LIN {X 0,Y 310.097,Z 794.889,A -85,B 0,C 180,E1 -20725.805,E2 -20725.805} C_VEL
LIN {X 0,Y 313.218,Z 774.353,A -85,B 0,C 180,E1 -20728.091,E2 -20728.091} C_VEL
LIN {X 0,Y 316.543,Z 751.825,A -85,B 0,C 180,E1 -20730.149,E2 -20730.149} C_VEL
LIN {X 0,Y 319.689,Z 728.685,A -85,B 0,C 180,E1 -20731.857,E2 -20731.857} C_VEL
LIN {X 0,Y 322.597,Z 704.405,A -85,B 0,C 180,E1 -20733.252,E2 -20733.252} C_VEL
LIN {X 0,Y 324.402,Z 688.186,A -85,B 0,C 180,E1 -20734.016,E2 -20734.016} C_VEL
LIN {X 0,Y 325.636,Z 688.059,A -85,B 0,C 180,E1 -20734.348,E2 -20734.348} C_VEL
LIN {X 0,Y 327.891,Z 685.502,A -85,B 0,C 180,E1 -20734.741,E2 -20734.741} C_VEL
LIN {X 0,Y 331.75,Z 678.48,A -85,B 0,C 180,E1 -20735.173,E2 -20735.173} C_VEL
LIN {X 0,Y 336.333,Z 667.667,A -85,B 0,C 180,E1 -20735.483,E2 -20735.483} C_VEL
LIN {X 0,Y 339.475,Z 663.92,A -85,B 0,C 180,E1 -20735.988,E2 -20735.988} C_VEL
LIN {X 0,Y 343.394,Z 656.895,A -85,B 0,C 180,E1 -20736.429,E2 -20736.429} C_VEL
LIN {X 0,Y 348.297,Z 645.248,A -85,B 0,C 180,E1 -20736.772,E2 -20736.772} C_VEL
LIN {X 0,Y 349.24,Z 643.212,A -85,B 0,C 180,E1 -20736.856,E2 -20736.856} C_VEL
LIN {X 0,Y 353.089,Z 637.648,A -85,B 0,C 180,E1 -20737.379,E2 -20737.379} C_VEL
LIN {X 0,Y 357.645,Z 628.586,A -85,B 0,C 180,E1 -20737.818,E2 -20737.818} C_VEL
LIN {X 0,Y 363.002,Z 615.103,A -85,B 0,C 180,E1 -20738.174,E2 -20738.174} C_VEL
LIN {X 0,Y 367.492,Z 607.691,A -85,B 0,C 180,E1 -20738.703,E2 -20738.703} C_VEL
LIN {X 0,Y 372.393,Z 596.823,A -85,B 0,C 180,E1 -20739.123,E2 -20739.123} C_VEL
LIN {X 0,Y 375.613,Z 588.328,A -85,B 0,C 180,E1 -20739.332,E2 -20739.332} C_VEL
LIN {X 0,Y 368.648,Z 640.972,A -85,B 0,C 180,E1 -20740.837,E2 -20740.837} C_VEL
LIN {X 0,Y 363.114,Z 683.795,A -85,B 0,C 180,E1 -20742.409,E2 -20742.409} C_VEL
LIN {X 0,Y 360.052,Z 705.878,A -85,B 0,C 180,E1 -20743.431,E2 -20743.431} C_VEL
LIN {X 0,Y 356.301,Z 726.402,A -85,B 0,C 180,E1 -20744.651,E2 -20744.651} C_VEL
LIN {X 0,Y 351.864,Z 746.01,A -85,B 0,C 180,E1 -20746.102,E2 -20746.102} C_VEL
LIN {X 0,Y 346.634,Z 765.549,A -85,B 0,C 180,E1 -20747.881,E2 -20747.881} C_VEL
LIN {X 0,Y 340.825,Z 784.337,A -85,B 0,C 180,E1 -20749.97,E2 -20749.97} C_VEL
LIN {X 0,Y 334.834,Z 801.656,A -85,B 0,C 180,E1 -20752.312,E2 -20752.312} C_VEL
LIN {X 0,Y 328.814,Z 817.581,A -85,B 0,C 180,E1 -20754.919,E2 -20754.919} C_VEL
LIN {X 0,Y 322.895,Z 832.224,A -85,B 0,C 180,E1 -20757.817,E2 -20757.817} C_VEL
LIN {X 0,Y 317.342,Z 845.359,A -85,B 0,C 180,E1 -20760.972,E2 -20760.972} C_VEL
LIN {X 0,Y 312.298,Z 857,A -85,B 0,C 180,E1 -20764.391,E2 -20764.391} C_VEL
LIN {X 0,Y 307.902,Z 867.134,A -85,B 0,C 180,E1 -20768.071,E2 -20768.071} C_VEL
LIN {X 0,Y 304.295,Z 875.703,A -85,B 0,C 180,E1 -20772.008,E2 -20772.008} C_VEL
LIN {X 0,Y 301.659,Z 882.344,A -85,B 0,C 180,E1 -20775.997,E2 -20775.997} C_VEL
LIN {X 0,Y 299.834,Z 887.403,A -85,B 0,C 180,E1 -20780.208,E2 -20780.208} C_VEL
LIN {X 0,Y 298.86,Z 890.521,A -85,B 0,C 180,E1 -20784.239,E2 -20784.239} C_VEL
LIN {X 0,Y 298.446,Z 892.023,A -85,B 0,C 180,E1 -20788.08,E2 -20788.08} C_VEL
LIN {X 0,Y 298.441,Z 892.036,A -85,B 0,C 180,E1 -20791.92,E2 -20791.92} C_VEL
LIN {X 0,Y 298.847,Z 890.585,A -85,B 0,C 180,E1 -20795.761,E2 -20795.761} C_VEL
LIN {X 0,Y 299.808,Z 887.52,A -85,B 0,C 180,E1 -20799.793,E2 -20799.793} C_VEL
LIN {X 0,Y 301.515,Z 882.791,A -85,B 0,C 180,E1 -20803.814,E2 -20803.814} C_VEL
LIN {X 0,Y 303.952,Z 876.657,A -85,B 0,C 180,E1 -20807.616,E2 -20807.616} C_VEL
LIN {X 0,Y 307.265,Z 868.804,A -85,B 0,C 180,E1 -20811.375,E2 -20811.375} C_VEL
LIN {X 0,Y 311.499,Z 859.044,A -85,B 0,C 180,E1 -20815.069,E2 -20815.069} C_VEL
LIN {X 0,Y 316.674,Z 847.142,A -85,B 0,C 180,E1 -20818.681,E2 -20818.681} C_VEL
LIN {X 0,Y 322.136,Z 834.333,A -85,B 0,C 180,E1 -20821.848,E2 -20821.848} C_VEL
LIN {X 0,Y 327.967,Z 820.047,A -85,B 0,C 180,E1 -20824.758,E2 -20824.758} C_VEL
LIN {X 0,Y 334.223,Z 803.699,A -85,B 0,C 180,E1 -20827.503,E2 -20827.503} C_VEL
LIN {X 0,Y 339.242,Z 789.378,A -85,B 0,C 180,E1 -20829.505,E2 -20829.505} C_VEL
LIN {X 0,Y 340.475,Z 783.625,A -85,B 0,C 180,E1 -20830.359,E2 -20830.359} C_VEL
LIN {X 0,Y 340.769,Z 769.373,A -85,B 0,C 180,E1 -20832.726,E2 -20832.726} C_VEL
LIN {X 0,Y 341.959,Z 763.048,A -85,B 0,C 180,E1 -20833.483,E2 -20833.483} C_VEL
LIN {X 0,Y 346.995,Z 744.339,A -85,B 0,C 180,E1 -20835.143,E2 -20835.143} C_VEL
LIN {X 0,Y 351.352,Z 725.232,A -85,B 0,C 180,E1 -20836.526,E2 -20836.526} C_VEL
LIN {X 0,Y 355.11,Z 704.688,A -85,B 0,C 180,E1 -20837.724,E2 -20837.724} C_VEL
LIN {X 0,Y 358.615,Z 679.329,A -85,B 0,C 180,E1 -20838.859,E2 -20838.859} C_VEL
LIN {X 0,Y 364.283,Z 637.626,A -85,B 0,C 180,E1 -20840.362,E2 -20840.362} C_VEL
LIN {X 0,Y 371.135,Z 586.782,A -85,B 0,C 180,E1 -20841.799,E2 -20841.799} C_VEL
LIN {X 0,Y 377.109,Z 533.395,A -85,B 0,C 180,E1 -20843.058,E2 -20843.058} C_VEL
LIN {X 0,Y 381.368,Z 483.071,A -85,B 0,C 180,E1 -20844.053,E2 -20844.053} C_VEL
LIN {X 0,Y 384.825,Z 436.662,A -85,B 0,C 180,E1 -20844.887,E2 -20844.887} C_VEL
LIN {X 0,Y 391.487,Z 407.522,A -85,B 0,C 180,E1 -20845.872,E2 -20845.872} C_VEL
LIN {X 0,Y 386.519,Z 392.199,A -85,B 0,C 180,E1 -20848.67,E2 -20848.67} C_VEL
LIN {X 0,Y 381.381,Z 378.048,A -85,B 0,C 180,E1 -20851.67,E2 -20851.67} C_VEL
LIN {X 0,Y 376.23,Z 365.361,A -85,B 0,C 180,E1 -20854.835,E2 -20854.835} C_VEL
LIN {X 0,Y 371.348,Z 354.346,A -85,B 0,C 180,E1 -20858.104,E2 -20858.104} C_VEL
LIN {X 0,Y 367.077,Z 345.55,A -85,B 0,C 180,E1 -20861.251,E2 -20861.251} C_VEL
LIN {X 0,Y 364.606,Z 340.77,A -85,B 0,C 180,E1 -20863.265,E2 -20863.265} C_VEL
LIN {X 0,Y 362.517,Z 336.712,A -85,B 0,C 180,E1 -20865.137,E2 -20865.137} C_VEL
LIN {X 0,Y 360.35,Z 332.462,A -85,B 0,C 180,E1 -20867.419,E2 -20867.419} C_VEL
LIN {X 0,Y 357.865,Z 327.689,A -85,B 0,C 180,E1 -20870.511,E2 -20870.511} C_VEL
LIN {X 0,Y 355.935,Z 324.353,A -85,B 0,C 180,E1 -20873.71,E2 -20873.71} C_VEL
LIN {X 0,Y 355.5,Z 322.634,A -85,B 0,C 180,E1 -20874.998,E2 -20874.998} C_VEL
LIN {X 0,Y 354.47,Z 320.986,A -85,B 0,C 180,E1 -20881.455,E2 -20881.455} C_VEL
LIN {X 0,Y 355.671,Z 321.876,A -85,B 0,C 180,E1 -20885.971,E2 -20885.971} C_VEL
LIN {X 0,Y 357.257,Z 323.157,A -85,B 0,C 180,E1 -20888.449,E2 -20888.449} C_VEL
LIN {X 0,Y 359.098,Z 335.798,A -85,B 0,C 180,E1 -20892.871,E2 -20892.871} C_VEL
LIN {X 0,Y 362.564,Z 349.288,A -85,B 0,C 180,E1 -20896.87,E2 -20896.87} C_VEL
LIN {X 0,Y 369.014,Z 369.011,A -85,B 0,C 180,E1 -20901.791,E2 -20901.791} C_VEL
LIN {X 0,Y 372.901,Z 379.636,A -85,B 0,C 180,E1 -20904.052,E2 -20904.052} C_VEL
LIN {X 0,Y 380.695,Z 402.746,A -85,B 0,C 180,E1 -20908.065,E2 -20908.065} C_VEL
LIN {X 0,Y 381.092,Z 404.189,A -85,B 0,C 180,E1 -20908.265,E2 -20908.265} C_VEL
LIN {X 0,Y 363.956,Z 554.058,A -85,B 0,C 180,E1 -20912.157,E2 -20912.157} C_VEL
LIN {X 0,Y 358.565,Z 611.238,A -85,B 0,C 180,E1 -20913.592,E2 -20913.592} C_VEL
LIN {X 0,Y 355.678,Z 653.164,A -85,B 0,C 180,E1 -20914.491,E2 -20914.491} C_VEL
LIN {X 0,Y 352.117,Z 687.641,A -85,B 0,C 180,E1 -20915.473,E2 -20915.473} C_VEL
LIN {X 0,Y 347.408,Z 721.446,A -85,B 0,C 180,E1 -20916.703,E2 -20916.703} C_VEL
LIN {X 0,Y 342.681,Z 750.705,A -85,B 0,C 180,E1 -20918.083,E2 -20918.083} C_VEL
LIN {X 0,Y 337.211,Z 780.861,A -85,B 0,C 180,E1 -20919.828,E2 -20919.828} C_VEL
LIN {X 0,Y 331.507,Z 809.252,A -85,B 0,C 180,E1 -20921.841,E2 -20921.841} C_VEL
LIN {X 0,Y 327.245,Z 827.893,A -85,B 0,C 180,E1 -20923.475,E2 -20923.475} C_VEL
LIN {X 0,Y 322.518,Z 845.852,A -85,B 0,C 180,E1 -20925.396,E2 -20925.396} C_VEL
LIN {X 0,Y 317.602,Z 862.404,A -85,B 0,C 180,E1 -20927.523,E2 -20927.523} C_VEL
LIN {X 0,Y 312.385,Z 878.87,A -85,B 0,C 180,E1 -20930.076,E2 -20930.076} C_VEL
LIN {X 0,Y 307.204,Z 894.344,A -85,B 0,C 180,E1 -20932.977,E2 -20932.977} C_VEL
LIN {X 0,Y 302.284,Z 908.668,A -85,B 0,C 180,E1 -20936.241,E2 -20936.241} C_VEL
LIN {X 0,Y 297.991,Z 921.531,A -85,B 0,C 180,E1 -20939.781,E2 -20939.781} C_VEL
LIN {X 0,Y 294.466,Z 932.94,A -85,B 0,C 180,E1 -20943.588,E2 -20943.588} C_VEL
LIN {X 0,Y 291.816,Z 942.875,A -85,B 0,C 180,E1 -20947.69,E2 -20947.69} C_VEL
LIN {X 0,Y 290.161,Z 951.193,A -85,B 0,C 180,E1 -20952.007,E2 -20952.007} C_VEL
LIN {X 0,Y 289.494,Z 957.489,A -85,B 0,C 180,E1 -20956.213,E2 -20956.213} C_VEL
LIN {X 0,Y 289.553,Z 962.147,A -85,B 0,C 180,E1 -20960.459,E2 -20960.459} C_VEL
LIN {X 0,Y 289.9,Z 965.745,A -85,B 0,C 180,E1 -20964.657,E2 -20964.657} C_VEL
LIN {X 0,Y 290.044,Z 968.016,A -85,B 0,C 180,E1 -20968.222,E2 -20968.222} C_VEL
LIN {X 0,Y 289.94,Z 968.994,A -85,B 0,C 180,E1 -20971.383,E2 -20971.383} C_VEL
LIN {X 0,Y 289.558,Z 968.983,A -85,B 0,C 180,E1 -20974.754,E2 -20974.754} C_VEL
LIN {X 0,Y 289.099,Z 967.8,A -85,B 0,C 180,E1 -20978.553,E2 -20978.553} C_VEL
LIN {X 0,Y 288.987,Z 964.607,A -85,B 0,C 180,E1 -20983.404,E2 -20983.404} C_VEL
LIN {X 0,Y 289.757,Z 960.148,A -85,B 0,C 180,E1 -20987.886,E2 -20987.886} C_VEL
LIN {X 0,Y 292.21,Z 953.138,A -85,B 0,C 180,E1 -20993.173,E2 -20993.173} C_VEL
LIN {X 0,Y 296.428,Z 944.613,A -85,B 0,C 180,E1 -20998.18,E2 -20998.18} C_VEL
LIN {X 0,Y 303.398,Z 933.28,A -85,B 0,C 180,E1 -21003.509,E2 -21003.509} C_VEL
LIN {X 0,Y 312.593,Z 920.465,A -85,B 0,C 180,E1 -21008.401,E2 -21008.401} C_VEL
LIN {X 0,Y 324.233,Z 905.701,A -85,B 0,C 180,E1 -21012.964,E2 -21012.964} C_VEL
LIN {X 0,Y 338.331,Z 889.038,A -85,B 0,C 180,E1 -21017.133,E2 -21017.133} C_VEL
LIN {X 0,Y 354.739,Z 870.663,A -85,B 0,C 180,E1 -21020.817,E2 -21020.817} C_VEL
LIN {X 0,Y 365.018,Z 859.44,A -85,B 0,C 180,E1 -21022.699,E2 -21022.699} C_VEL
LIN {X 0,Y 349.209,Z 872.446,A -85,B 0,C 180,E1 -21025.662,E2 -21025.662} C_VEL
LIN {X 0,Y 335.594,Z 883.653,A -85,B 0,C 180,E1 -21028.972,E2 -21028.972} C_VEL
LIN {X 0,Y 324.384,Z 892.704,A -85,B 0,C 180,E1 -21032.46,E2 -21032.46} C_VEL
LIN {X 0,Y 315.292,Z 899.629,A -85,B 0,C 180,E1 -21036.051,E2 -21036.051} C_VEL
LIN {X 0,Y 308.049,Z 904.537,A -85,B 0,C 180,E1 -21039.677,E2 -21039.677} C_VEL
LIN {X 0,Y 302.172,Z 907.645,A -85,B 0,C 180,E1 -21043.467,E2 -21043.467} C_VEL
LIN {X 0,Y 297.811,Z 908.844,A -85,B 0,C 180,E1 -21047.197,E2 -21047.197} C_VEL
LIN {X 0,Y 294.664,Z 908.287,A -85,B 0,C 180,E1 -21050.917,E2 -21050.917} C_VEL
LIN {X 0,Y 292.468,Z 905.923,A -85,B 0,C 180,E1 -21054.704,E2 -21054.704} C_VEL
LIN {X 0,Y 291.159,Z 901.801,A -85,B 0,C 180,E1 -21058.426,E2 -21058.426} C_VEL
LIN {X 0,Y 290.513,Z 895.812,A -85,B 0,C 180,E1 -21062.17,E2 -21062.17} C_VEL
LIN {X 0,Y 290.44,Z 888.231,A -85,B 0,C 180,E1 -21065.769,E2 -21065.769} C_VEL
LIN {X 0,Y 290.873,Z 878.851,A -85,B 0,C 180,E1 -21069.298,E2 -21069.298} C_VEL
LIN {X 0,Y 291.811,Z 867.931,A -85,B 0,C 180,E1 -21072.668,E2 -21072.668} C_VEL
LIN {X 0,Y 293.234,Z 855.611,A -85,B 0,C 180,E1 -21075.83,E2 -21075.83} C_VEL
LIN {X 0,Y 295.081,Z 841.982,A -85,B 0,C 180,E1 -21078.779,E2 -21078.779} C_VEL
LIN {X 0,Y 297.464,Z 826.09,A -85,B 0,C 180,E1 -21081.7,E2 -21081.7} C_VEL
LIN {X 0,Y 300.213,Z 808.748,A -85,B 0,C 180,E1 -21084.393,E2 -21084.393} C_VEL
LIN {X 0,Y 303.242,Z 789.904,A -85,B 0,C 180,E1 -21086.855,E2 -21086.855} C_VEL
LIN {X 0,Y 306.442,Z 769.276,A -85,B 0,C 180,E1 -21089.09,E2 -21089.09} C_VEL
LIN {X 0,Y 309.807,Z 746.584,A -85,B 0,C 180,E1 -21091.091,E2 -21091.091} C_VEL
LIN {X 0,Y 313.021,Z 722.706,A -85,B 0,C 180,E1 -21092.782,E2 -21092.782} C_VEL
LIN {X 0,Y 314.397,Z 711.79,A -85,B 0,C 180,E1 -21093.435,E2 -21093.435} C_VEL
LIN {X 0,Y 315.558,Z 711.842,A -85,B 0,C 180,E1 -21093.787,E2 -21093.787} C_VEL
LIN {X 0,Y 317.977,Z 709.611,A -85,B 0,C 180,E1 -21094.255,E2 -21094.255} C_VEL
LIN {X 0,Y 321.775,Z 703.882,A -85,B 0,C 180,E1 -21094.738,E2 -21094.738} C_VEL
LIN {X 0,Y 326.016,Z 695.125,A -85,B 0,C 180,E1 -21095.091,E2 -21095.091} C_VEL
LIN {X 0,Y 329.867,Z 690.849,A -85,B 0,C 180,E1 -21095.724,E2 -21095.724} C_VEL
LIN {X 0,Y 333.975,Z 683.923,A -85,B 0,C 180,E1 -21096.196,E2 -21096.196} C_VEL
LIN {X 0,Y 338.441,Z 674.02,A -85,B 0,C 180,E1 -21096.514,E2 -21096.514} C_VEL
LIN {X 0,Y 339.39,Z 672.118,A -85,B 0,C 180,E1 -21096.6,E2 -21096.6} C_VEL
LIN {X 0,Y 343.392,Z 666.592,A -85,B 0,C 180,E1 -21097.145,E2 -21097.145} C_VEL
LIN {X 0,Y 348.05,Z 657.692,A -85,B 0,C 180,E1 -21097.589,E2 -21097.589} C_VEL
LIN {X 0,Y 352.501,Z 647.411,A -85,B 0,C 180,E1 -21097.888,E2 -21097.888} C_VEL
LIN {X 0,Y 357.058,Z 640.454,A -85,B 0,C 180,E1 -21098.439,E2 -21098.439} C_VEL
LIN {X 0,Y 362.014,Z 630.337,A -85,B 0,C 180,E1 -21098.87,E2 -21098.87} C_VEL
LIN {X 0,Y 366.643,Z 618.897,A -85,B 0,C 180,E1 -21099.159,E2 -21099.159} C_VEL
LIN {X 0,Y 360.03,Z 667.651,A -85,B 0,C 180,E1 -21100.794,E2 -21100.794} C_VEL
LIN {X 0,Y 355.595,Z 700.826,A -85,B 0,C 180,E1 -21102.189,E2 -21102.189} C_VEL
LIN {X 0,Y 351.844,Z 722.205,A -85,B 0,C 180,E1 -21103.388,E2 -21103.388} C_VEL
LIN {X 0,Y 347.315,Z 742.561,A -85,B 0,C 180,E1 -21104.826,E2 -21104.826} C_VEL
LIN {X 0,Y 342.182,Z 761.879,A -85,B 0,C 180,E1 -21106.516,E2 -21106.516} C_VEL
LIN {X 0,Y 336.449,Z 780.451,A -85,B 0,C 180,E1 -21108.497,E2 -21108.497} C_VEL
LIN {X 0,Y 330.364,Z 797.932,A -85,B 0,C 180,E1 -21110.76,E2 -21110.76} C_VEL
LIN {X 0,Y 324.065,Z 814.382,A -85,B 0,C 180,E1 -21113.343,E2 -21113.343} C_VEL
LIN {X 0,Y 317.926,Z 829.258,A -85,B 0,C 180,E1 -21116.174,E2 -21116.174} C_VEL
LIN {X 0,Y 311.925,Z 843.014,A -85,B 0,C 180,E1 -21119.357,E2 -21119.357} C_VEL
LIN {X 0,Y 306.423,Z 855.219,A -85,B 0,C 180,E1 -21122.817,E2 -21122.817} C_VEL
LIN {X 0,Y 301.577,Z 865.858,A -85,B 0,C 180,E1 -21126.555,E2 -21126.555} C_VEL
LIN {X 0,Y 297.526,Z 874.902,A -85,B 0,C 180,E1 -21130.567,E2 -21130.567} C_VEL
LIN {X 0,Y 294.517,Z 881.994,A -85,B 0,C 180,E1 -21134.644,E2 -21134.644} C_VEL
LIN {X 0,Y 292.358,Z 887.482,A -85,B 0,C 180,E1 -21138.958,E2 -21138.958} C_VEL
LIN {X 0,Y 291.105,Z 891.11,A -85,B 0,C 180,E1 -21143.293,E2 -21143.293} C_VEL
LIN {X 0,Y 290.551,Z 892.885,A -85,B 0,C 180,E1 -21147.436,E2 -21147.436} C_VEL
LIN {X 0,Y 290.477,Z 893.097,A -85,B 0,C 180,E1 -21151.381,E2 -21151.381} C_VEL
LIN {X 0,Y 290.873,Z 891.794,A -85,B 0,C 180,E1 -21155.523,E2 -21155.523} C_VEL
LIN {X 0,Y 291.835,Z 888.902,A -85,B 0,C 180,E1 -21159.665,E2 -21159.665} C_VEL
LIN {X 0,Y 293.569,Z 884.354,A -85,B 0,C 180,E1 -21163.793,E2 -21163.793} C_VEL
LIN {X 0,Y 296.202,Z 878.044,A -85,B 0,C 180,E1 -21167.89,E2 -21167.89} C_VEL
LIN {X 0,Y 299.836,Z 869.83,A -85,B 0,C 180,E1 -21171.931,E2 -21171.931} C_VEL
LIN {X 0,Y 304.281,Z 860.081,A -85,B 0,C 180,E1 -21175.706,E2 -21175.706} C_VEL
LIN {X 0,Y 309.693,Z 848.18,A -85,B 0,C 180,E1 -21179.39,E2 -21179.39} C_VEL
LIN {X 0,Y 315.388,Z 835.383,A -85,B 0,C 180,E1 -21182.613,E2 -21182.613} C_VEL
LIN {X 0,Y 321.456,Z 821.111,A -85,B 0,C 180,E1 -21185.568,E2 -21185.568} C_VEL
LIN {X 0,Y 327.943,Z 804.743,A -85,B 0,C 180,E1 -21188.35,E2 -21188.35} C_VEL
LIN {X 0,Y 334.1,Z 787.79,A -85,B 0,C 180,E1 -21190.725,E2 -21190.725} C_VEL
LIN {X 0,Y 339.952,Z 769.852,A -85,B 0,C 180,E1 -21192.799,E2 -21192.799} C_VEL
LIN {X 0,Y 341.959,Z 763.048,A -85,B 0,C 180,E1 -21193.483,E2 -21193.483} C_VEL
LIN {X 0,Y 343.111,Z 756.729,A -85,B 0,C 180,E1 -21194.213,E2 -21194.213} C_VEL
LIN {X 0,Y 343.287,Z 740.949,A -85,B 0,C 180,E1 -21196.295,E2 -21196.295} C_VEL
LIN {X 0,Y 344.169,Z 734.277,A -85,B 0,C 180,E1 -21196.932,E2 -21196.932} C_VEL
LIN {X 0,Y 348.496,Z 713.392,A -85,B 0,C 180,E1 -21198.268,E2 -21198.268} C_VEL
LIN {X 0,Y 351.931,Z 691.641,A -85,B 0,C 180,E1 -21199.351,E2 -21199.351} C_VEL
LIN {X 0,Y 357.689,Z 649.532,A -85,B 0,C 180,E1 -21200.974,E2 -21200.974} C_VEL
LIN {X 0,Y 364.593,Z 600.878,A -85,B 0,C 180,E1 -21202.435,E2 -21202.435} C_VEL
LIN {X 0,Y 370.767,Z 550.378,A -85,B 0,C 180,E1 -21203.692,E2 -21203.692} C_VEL
LIN {X 0,Y 375.515,Z 499.905,A -85,B 0,C 180,E1 -21204.738,E2 -21204.738} C_VEL
LIN {X 0,Y 380.163,Z 439.411,A -85,B 0,C 180,E1 -21205.836,E2 -21205.836} C_VEL
LIN {X 0,Y 386.666,Z 411.148,A -85,B 0,C 180,E1 -21206.777,E2 -21206.777} C_VEL
LIN {X 0,Y 381.926,Z 396.352,A -85,B 0,C 180,E1 -21209.563,E2 -21209.563} C_VEL
LIN {X 0,Y 376.863,Z 382.161,A -85,B 0,C 180,E1 -21212.677,E2 -21212.677} C_VEL
LIN {X 0,Y 372.149,Z 370.419,A -85,B 0,C 180,E1 -21215.727,E2 -21215.727} C_VEL
LIN {X 0,Y 367.922,Z 360.719,A -85,B 0,C 180,E1 -21218.685,E2 -21218.685} C_VEL
LIN {X 0,Y 364.04,Z 352.331,A -85,B 0,C 180,E1 -21221.753,E2 -21221.753} C_VEL
LIN {X 0,Y 361.674,Z 347.588,A -85,B 0,C 180,E1 -21223.786,E2 -21223.786} C_VEL
LIN {X 0,Y 359.895,Z 343.923,A -85,B 0,C 180,E1 -21225.52,E2 -21225.52} C_VEL
LIN {X 0,Y 357.988,Z 339.875,A -85,B 0,C 180,E1 -21227.744,E2 -21227.744} C_VEL
LIN {X 0,Y 355.585,Z 335.237,A -85,B 0,C 180,E1 -21230.777,E2 -21230.777} C_VEL
LIN {X 0,Y 353.736,Z 331.636,A -85,B 0,C 180,E1 -21234.159,E2 -21234.159} C_VEL
LIN {X 0,Y 353.406,Z 330.304,A -85,B 0,C 180,E1 -21235.294,E2 -21235.294} C_VEL
LIN {X 0,Y 352.685,Z 328.775,A -85,B 0,C 180,E1 -21241.625,E2 -21241.625} C_VEL
LIN {X 0,Y 354.065,Z 329.807,A -85,B 0,C 180,E1 -21246.323,E2 -21246.323} C_VEL
LIN {X 0,Y 355.236,Z 330.811,A -85,B 0,C 180,E1 -21248.172,E2 -21248.172} C_VEL
LIN {X 0,Y 356.963,Z 342.871,A -85,B 0,C 180,E1 -21252.374,E2 -21252.374} C_VEL
LIN {X 0,Y 360.086,Z 356.086,A -85,B 0,C 180,E1 -21256.329,E2 -21256.329} C_VEL
LIN {X 0,Y 366.35,Z 375.856,A -85,B 0,C 180,E1 -21261.285,E2 -21261.285} C_VEL
LIN {X 0,Y 369.886,Z 385.971,A -85,B 0,C 180,E1 -21263.457,E2 -21263.457} C_VEL
LIN {X 0,Y 376.95,Z 407.665,A -85,B 0,C 180,E1 -21267.271,E2 -21267.271} C_VEL
LIN {X 0,Y 356.204,Z 579.083,A -85,B 0,C 180,E1 -21271.835,E2 -21271.835} C_VEL
LIN {X 0,Y 351.392,Z 648.87,A -85,B 0,C 180,E1 -21273.325,E2 -21273.325} C_VEL
LIN {X 0,Y 347.833,Z 683.011,A -85,B 0,C 180,E1 -21274.279,E2 -21274.279} C_VEL
LIN {X 0,Y 343.149,Z 716.179,A -85,B 0,C 180,E1 -21275.459,E2 -21275.459} C_VEL
LIN {X 0,Y 338.014,Z 746.973,A -85,B 0,C 180,E1 -21276.867,E2 -21276.867} C_VEL
LIN {X 0,Y 332.497,Z 776.814,A -85,B 0,C 180,E1 -21278.567,E2 -21278.567} C_VEL
LIN {X 0,Y 326.517,Z 805.796,A -85,B 0,C 180,E1 -21280.585,E2 -21280.585} C_VEL
LIN {X 0,Y 322.047,Z 824.838,A -85,B 0,C 180,E1 -21282.227,E2 -21282.227} C_VEL
LIN {X 0,Y 316.988,Z 843.135,A -85,B 0,C 180,E1 -21284.155,E2 -21284.155} C_VEL
LIN {X 0,Y 311.435,Z 861.14,A -85,B 0,C 180,E1 -21286.475,E2 -21286.475} C_VEL
LIN {X 0,Y 305.778,Z 878.186,A -85,B 0,C 180,E1 -21289.156,E2 -21289.156} C_VEL
LIN {X 0,Y 300.361,Z 893.477,A -85,B 0,C 180,E1 -21292.089,E2 -21292.089} C_VEL
LIN {X 0,Y 295.216,Z 907.713,A -85,B 0,C 180,E1 -21295.39,E2 -21295.39} C_VEL
LIN {X 0,Y 290.74,Z 920.364,A -85,B 0,C 180,E1 -21298.945,E2 -21298.945} C_VEL
LIN {X 0,Y 286.97,Z 931.798,A -85,B 0,C 180,E1 -21302.842,E2 -21302.842} C_VEL
LIN {X 0,Y 284.132,Z 941.659,A -85,B 0,C 180,E1 -21307.007,E2 -21307.007} C_VEL
LIN {X 0,Y 282.324,Z 949.983,A -85,B 0,C 180,E1 -21311.413,E2 -21311.413} C_VEL
LIN {X 0,Y 281.545,Z 956.442,A -85,B 0,C 180,E1 -21315.824,E2 -21315.824} C_VEL
LIN {X 0,Y 281.547,Z 960.921,A -85,B 0,C 180,E1 -21319.979,E2 -21319.979} C_VEL
LIN {X 0,Y 282.01,Z 964.446,A -85,B 0,C 180,E1 -21324.711,E2 -21324.711} C_VEL
LIN {X 0,Y 282.157,Z 966.76,A -85,B 0,C 180,E1 -21328.376,E2 -21328.376} C_VEL
LIN {X 0,Y 281.994,Z 967.796,A -85,B 0,C 180,E1 -21331.829,E2 -21331.829} C_VEL
LIN {X 0,Y 281.58,Z 967.758,A -85,B 0,C 180,E1 -21335.298,E2 -21335.298} C_VEL
LIN {X 0,Y 281.082,Z 966.455,A -85,B 0,C 180,E1 -21339.418,E2 -21339.418} C_VEL
LIN {X 0,Y 281.08,Z 963.184,A -85,B 0,C 180,E1 -21344.419,E2 -21344.419} C_VEL
LIN {X 0,Y 282.123,Z 958.691,A -85,B 0,C 180,E1 -21349.03,E2 -21349.03} C_VEL
LIN {X 0,Y 285.023,Z 951.705,A -85,B 0,C 180,E1 -21354.454,E2 -21354.454} C_VEL
LIN {X 0,Y 290.041,Z 942.875,A -85,B 0,C 180,E1 -21359.764,E2 -21359.764} C_VEL
LIN {X 0,Y 297.987,Z 931.43,A -85,B 0,C 180,E1 -21365.25,E2 -21365.25} C_VEL
LIN {X 0,Y 308.228,Z 918.66,A -85,B 0,C 180,E1 -21370.208,E2 -21370.208} C_VEL
LIN {X 0,Y 320.962,Z 904.077,A -85,B 0,C 180,E1 -21374.754,E2 -21374.754} C_VEL
LIN {X 0,Y 336.752,Z 887.173,A -85,B 0,C 180,E1 -21378.989,E2 -21378.989} C_VEL
LIN {X 0,Y 353.463,Z 870.171,A -85,B 0,C 180,E1 -21382.38,E2 -21382.38} C_VEL
LIN {X 0,Y 355.449,Z 868.133,A -85,B 0,C 180,E1 -21382.756,E2 -21382.756} C_VEL
LIN {X 0,Y 339.797,Z 879.829,A -85,B 0,C 180,E1 -21385.803,E2 -21385.803} C_VEL
LIN {X 0,Y 326.256,Z 889.867,A -85,B 0,C 180,E1 -21389.215,E2 -21389.215} C_VEL
LIN {X 0,Y 315.116,Z 897.821,A -85,B 0,C 180,E1 -21392.811,E2 -21392.811} C_VEL
LIN {X 0,Y 306.095,Z 903.73,A -85,B 0,C 180,E1 -21396.514,E2 -21396.514} C_VEL
LIN {X 0,Y 298.648,Z 907.843,A -85,B 0,C 180,E1 -21400.439,E2 -21400.439} C_VEL
LIN {X 0,Y 292.968,Z 909.937,A -85,B 0,C 180,E1 -21404.358,E2 -21404.358} C_VEL
LIN {X 0,Y 288.828,Z 910.181,A -85,B 0,C 180,E1 -21408.214,E2 -21408.214} C_VEL
LIN {X 0,Y 285.968,Z 908.753,A -85,B 0,C 180,E1 -21411.96,E2 -21411.96} C_VEL
LIN {X 0,Y 283.949,Z 905.358,A -85,B 0,C 180,E1 -21415.961,E2 -21415.961} C_VEL
LIN {X 0,Y 282.868,Z 900.293,A -85,B 0,C 180,E1 -21419.797,E2 -21419.797} C_VEL
LIN {X 0,Y 282.437,Z 893.734,A -85,B 0,C 180,E1 -21423.45,E2 -21423.45} C_VEL
LIN {X 0,Y 282.553,Z 885.362,A -85,B 0,C 180,E1 -21427.115,E2 -21427.115} C_VEL
LIN {X 0,Y 283.163,Z 875.563,A -85,B 0,C 180,E1 -21430.581,E2 -21430.581} C_VEL
LIN {X 0,Y 284.429,Z 862.976,A -85,B 0,C 180,E1 -21434.246,E2 -21434.246} C_VEL
LIN {X 0,Y 286.155,Z 849.601,A -85,B 0,C 180,E1 -21437.488,E2 -21437.488} C_VEL
LIN {X 0,Y 288.324,Z 834.796,A -85,B 0,C 180,E1 -21440.504,E2 -21440.504} C_VEL
LIN {X 0,Y 290.976,Z 818.009,A -85,B 0,C 180,E1 -21443.395,E2 -21443.395} C_VEL
LIN {X 0,Y 293.944,Z 799.899,A -85,B 0,C 180,E1 -21446.028,E2 -21446.028} C_VEL
LIN {X 0,Y 297.289,Z 779.355,A -85,B 0,C 180,E1 -21448.529,E2 -21448.529} C_VEL
LIN {X 0,Y 300.696,Z 757.667,A -85,B 0,C 180,E1 -21450.692,E2 -21450.692} C_VEL
LIN {X 0,Y 304.018,Z 734.908,A -85,B 0,C 180,E1 -21452.53,E2 -21452.53} C_VEL
LIN {X 0,Y 304.579,Z 731.096,A -85,B 0,C 180,E1 -21452.816,E2 -21452.816} C_VEL
LIN {X 0,Y 306.11,Z 730.891,A -85,B 0,C 180,E1 -21453.282,E2 -21453.282} C_VEL
LIN {X 0,Y 308.996,Z 728.323,A -85,B 0,C 180,E1 -21453.82,E2 -21453.82} C_VEL
LIN {X 0,Y 313.01,Z 722.831,A -85,B 0,C 180,E1 -21454.32,E2 -21454.32} C_VEL
LIN {X 0,Y 315.541,Z 718.67,A -85,B 0,C 180,E1 -21454.557,E2 -21454.557} C_VEL
LIN {X 0,Y 319.129,Z 715.537,A -85,B 0,C 180,E1 -21455.205,E2 -21455.205} C_VEL
LIN {X 0,Y 323.29,Z 709.874,A -85,B 0,C 180,E1 -21455.744,E2 -21455.744} C_VEL
LIN {X 0,Y 328.312,Z 700.656,A -85,B 0,C 180,E1 -21456.177,E2 -21456.177} C_VEL
LIN {X 0,Y 329.111,Z 699.455,A -85,B 0,C 180,E1 -21456.277,E2 -21456.277} C_VEL
LIN {X 0,Y 333.176,Z 694.404,A -85,B 0,C 180,E1 -21456.859,E2 -21456.859} C_VEL
LIN {X 0,Y 337.92,Z 686.155,A -85,B 0,C 180,E1 -21457.343,E2 -21457.343} C_VEL
LIN {X 0,Y 342.453,Z 676.446,A -85,B 0,C 180,E1 -21457.66,E2 -21457.66} C_VEL
LIN {X 0,Y 347.169,Z 669.599,A -85,B 0,C 180,E1 -21458.234,E2 -21458.234} C_VEL
LIN {X 0,Y 352.346,Z 659.543,A -85,B 0,C 180,E1 -21458.671,E2 -21458.671} C_VEL
LIN {X 0,Y 355.868,Z 651.493,A -85,B 0,C 180,E1 -21458.895,E2 -21458.895} C_VEL
LIN {X 0,Y 357.637,Z 649.135,A -85,B 0,C 180,E1 -21459.116,E2 -21459.116} C_VEL
LIN {X 0,Y 351.847,Z 691.074,A -85,B 0,C 180,E1 -21460.738,E2 -21460.738} C_VEL
LIN {X 0,Y 348.458,Z 712.778,A -85,B 0,C 180,E1 -21461.811,E2 -21461.811} C_VEL
LIN {X 0,Y 344.081,Z 734.017,A -85,B 0,C 180,E1 -21463.164,E2 -21463.164} C_VEL
LIN {X 0,Y 339.136,Z 753.596,A -85,B 0,C 180,E1 -21464.72,E2 -21464.72} C_VEL
LIN {X 0,Y 333.354,Z 772.976,A -85,B 0,C 180,E1 -21466.616,E2 -21466.616} C_VEL
LIN {X 0,Y 327.127,Z 791.223,A -85,B 0,C 180,E1 -21468.8,E2 -21468.8} C_VEL
LIN {X 0,Y 320.606,Z 808.342,A -85,B 0,C 180,E1 -21471.295,E2 -21471.295} C_VEL
LIN {X 0,Y 314.356,Z 823.41,A -85,B 0,C 180,E1 -21473.953,E2 -21473.953} C_VEL
LIN {X 0,Y 308.117,Z 837.495,A -85,B 0,C 180,E1 -21476.962,E2 -21476.962} C_VEL
LIN {X 0,Y 302.257,Z 850.138,A -85,B 0,C 180,E1 -21480.25,E2 -21480.25} C_VEL
LIN {X 0,Y 296.681,Z 861.846,A -85,B 0,C 180,E1 -21484.015,E2 -21484.015} C_VEL
LIN {X 0,Y 292.104,Z 871.467,A -85,B 0,C 180,E1 -21487.88,E2 -21487.88} C_VEL
LIN {X 0,Y 288.361,Z 879.551,A -85,B 0,C 180,E1 -21492.025,E2 -21492.025} C_VEL
LIN {X 0,Y 285.658,Z 885.743,A -85,B 0,C 180,E1 -21496.23,E2 -21496.23} C_VEL
LIN {X 0,Y 283.884,Z 890.175,A -85,B 0,C 180,E1 -21500.476,E2 -21500.476} C_VEL
LIN {X 0,Y 282.942,Z 892.841,A -85,B 0,C 180,E1 -21504.525,E2 -21504.525} C_VEL
LIN {X 0,Y 282.536,Z 894.107,A -85,B 0,C 180,E1 -21508.783,E2 -21508.783} C_VEL
LIN {X 0,Y 282.626,Z 893.861,A -85,B 0,C 180,E1 -21512.839,E2 -21512.839} C_VEL
LIN {X 0,Y 283.235,Z 892.063,A -85,B 0,C 180,E1 -21517.097,E2 -21517.097} C_VEL
LIN {X 0,Y 284.594,Z 888.422,A -85,B 0,C 180,E1 -21521.552,E2 -21521.552} C_VEL
LIN {X 0,Y 286.916,Z 882.914,A -85,B 0,C 180,E1 -21525.98,E2 -21525.98} C_VEL
LIN {X 0,Y 290.121,Z 875.798,A -85,B 0,C 180,E1 -21530.16,E2 -21530.16} C_VEL
LIN {X 0,Y 294.418,Z 866.728,A -85,B 0,C 180,E1 -21534.264,E2 -21534.264} C_VEL
LIN {X 0,Y 299.529,Z 856.058,A -85,B 0,C 180,E1 -21538.079,E2 -21538.079} C_VEL
LIN {X 0,Y 305.402,Z 843.624,A -85,B 0,C 180,E1 -21541.652,E2 -21541.652} C_VEL
LIN {X 0,Y 311.589,Z 830.016,A -85,B 0,C 180,E1 -21544.834,E2 -21544.834} C_VEL
LIN {X 0,Y 318.201,Z 814.584,A -85,B 0,C 180,E1 -21547.789,E2 -21547.789} C_VEL
LIN {X 0,Y 324.768,Z 797.965,A -85,B 0,C 180,E1 -21550.397,E2 -21550.397} C_VEL
LIN {X 0,Y 331.11,Z 780.235,A -85,B 0,C 180,E1 -21552.683,E2 -21552.683} C_VEL
LIN {X 0,Y 336.784,Z 762.36,A -85,B 0,C 180,E1 -21554.588,E2 -21554.588} C_VEL
LIN {X 0,Y 342.19,Z 742.493,A -85,B 0,C 180,E1 -21556.319,E2 -21556.319} C_VEL
LIN {X 0,Y 344.169,Z 734.277,A -85,B 0,C 180,E1 -21556.932,E2 -21556.932} C_VEL
LIN {X 0,Y 345.161,Z 727.504,A -85,B 0,C 180,E1 -21557.544,E2 -21557.544} C_VEL
LIN {X 0,Y 344.675,Z 710.571,A -85,B 0,C 180,E1 -21559.35,E2 -21559.35} C_VEL
LIN {X 0,Y 345.144,Z 703.415,A -85,B 0,C 180,E1 -21559.84,E2 -21559.84} C_VEL
LIN {X 0,Y 350.733,Z 664.574,A -85,B 0,C 180,E1 -21561.479,E2 -21561.479} C_VEL
LIN {X 0,Y 356.943,Z 622.303,A -85,B 0,C 180,E1 -21562.877,E2 -21562.877} C_VEL
LIN {X 0,Y 363.707,Z 572.195,A -85,B 0,C 180,E1 -21564.209,E2 -21564.209} C_VEL
LIN {X 0,Y 369.148,Z 521.87,A -85,B 0,C 180,E1 -21565.33,E2 -21565.33} C_VEL
LIN {X 0,Y 374.356,Z 456.234,A -85,B 0,C 180,E1 -21566.543,E2 -21566.543} C_VEL
LIN {X 0,Y 375.644,Z 442.026,A -85,B 0,C 180,E1 -21566.813,E2 -21566.813} C_VEL
LIN {X 0,Y 381.952,Z 414.888,A -85,B 0,C 180,E1 -21567.695,E2 -21567.695} C_VEL
LIN {X 0,Y 377.182,Z 399.775,A -85,B 0,C 180,E1 -21570.631,E2 -21570.631} C_VEL
LIN {X 0,Y 372.444,Z 386.352,A -85,B 0,C 180,E1 -21573.706,E2 -21573.706} C_VEL
LIN {X 0,Y 367.993,Z 374.96,A -85,B 0,C 180,E1 -21576.797,E2 -21576.797} C_VEL
LIN {X 0,Y 363.588,Z 364.648,A -85,B 0,C 180,E1 -21580.103,E2 -21580.103} C_VEL
LIN {X 0,Y 359.792,Z 356.235,A -85,B 0,C 180,E1 -21583.45,E2 -21583.45} C_VEL
LIN {X 0,Y 357.363,Z 351.267,A -85,B 0,C 180,E1 -21585.829,E2 -21585.829} C_VEL
LIN {X 0,Y 355.676,Z 347.381,A -85,B 0,C 180,E1 -21587.993,E2 -21587.993} C_VEL
LIN {X 0,Y 353.511,Z 342.934,A -85,B 0,C 180,E1 -21590.886,E2 -21590.886} C_VEL
LIN {X 0,Y 351.685,Z 339.321,A -85,B 0,C 180,E1 -21594.325,E2 -21594.325} C_VEL
LIN {X 0,Y 351.434,Z 338.035,A -85,B 0,C 180,E1 -21595.431,E2 -21595.431} C_VEL
LIN {X 0,Y 350.792,Z 336.546,A -85,B 0,C 180,E1 -21601.797,E2 -21601.797} C_VEL
LIN {X 0,Y 352.569,Z 337.811,A -85,B 0,C 180,E1 -21606.841,E2 -21606.841} C_VEL
LIN {X 0,Y 353.238,Z 338.552,A -85,B 0,C 180,E1 -21607.932,E2 -21607.932} C_VEL
LIN {X 0,Y 354.771,Z 350.186,A -85,B 0,C 180,E1 -21611.956,E2 -21611.956} C_VEL
LIN {X 0,Y 357.683,Z 362.885,A -85,B 0,C 180,E1 -21615.775,E2 -21615.775} C_VEL
LIN {X 0,Y 363.605,Z 382.359,A -85,B 0,C 180,E1 -21620.693,E2 -21620.693} C_VEL
LIN {X 0,Y 366.869,Z 392.296,A -85,B 0,C 180,E1 -21622.854,E2 -21622.854} C_VEL
LIN {X 0,Y 372.922,Z 411.537,A -85,B 0,C 180,E1 -21626.268,E2 -21626.268} C_VEL
LIN {X 0,Y 351.644,Z 581.817,A -85,B 0,C 180,E1 -21630.808,E2 -21630.808} C_VEL
LIN {X 0,Y 347.333,Z 643.921,A -85,B 0,C 180,E1 -21632.115,E2 -21632.115} C_VEL
LIN {X 0,Y 343.821,Z 677.097,A -85,B 0,C 180,E1 -21633.022,E2 -21633.022} C_VEL
LIN {X 0,Y 339.246,Z 709.541,A -85,B 0,C 180,E1 -21634.141,E2 -21634.141} C_VEL
LIN {X 0,Y 334.198,Z 739.62,A -85,B 0,C 180,E1 -21635.439,E2 -21635.439} C_VEL
LIN {X 0,Y 329.139,Z 766.452,A -85,B 0,C 180,E1 -21636.908,E2 -21636.908} C_VEL
LIN {X 0,Y 323.665,Z 792.898,A -85,B 0,C 180,E1 -21638.612,E2 -21638.612} C_VEL
LIN {X 0,Y 318.9,Z 813.963,A -85,B 0,C 180,E1 -21640.233,E2 -21640.233} C_VEL
LIN {X 0,Y 313.811,Z 833.029,A -85,B 0,C 180,E1 -21642.064,E2 -21642.064} C_VEL
LIN {X 0,Y 308.277,Z 851.263,A -85,B 0,C 180,E1 -21644.215,E2 -21644.215} C_VEL
LIN {X 0,Y 302.587,Z 868.119,A -85,B 0,C 180,E1 -21646.634,E2 -21646.634} C_VEL
LIN {X 0,Y 296.762,Z 884.18,A -85,B 0,C 180,E1 -21649.437,E2 -21649.437} C_VEL
LIN {X 0,Y 291.203,Z 898.921,A -85,B 0,C 180,E1 -21652.573,E2 -21652.573} C_VEL
LIN {X 0,Y 285.848,Z 912.994,A -85,B 0,C 180,E1 -21656.208,E2 -21656.208} C_VEL
LIN {X 0,Y 281.5,Z 924.876,A -85,B 0,C 180,E1 -21659.945,E2 -21659.945} C_VEL
LIN {X 0,Y 277.904,Z 935.632,A -85,B 0,C 180,E1 -21664.092,E2 -21664.092} C_VEL
LIN {X 0,Y 275.364,Z 944.751,A -85,B 0,C 180,E1 -21668.485,E2 -21668.485} C_VEL
LIN {X 0,Y 273.934,Z 952.193,A -85,B 0,C 180,E1 -21673.022,E2 -21673.022} C_VEL
LIN {X 0,Y 273.513,Z 957.825,A -85,B 0,C 180,E1 -21677.544,E2 -21677.544} C_VEL
LIN {X 0,Y 273.762,Z 961.703,A -85,B 0,C 180,E1 -21682.022,E2 -21682.022} C_VEL
LIN {X 0,Y 274.215,Z 964.141,A -85,B 0,C 180,E1 -21686.237,E2 -21686.237} C_VEL
LIN {X 0,Y 274.249,Z 965.886,A -85,B 0,C 180,E1 -21689.582,E2 -21689.582} C_VEL
LIN {X 0,Y 273.977,Z 966.635,A -85,B 0,C 180,E1 -21692.929,E2 -21692.929} C_VEL
LIN {X 0,Y 273.434,Z 966.354,A -85,B 0,C 180,E1 -21696.72,E2 -21696.72} C_VEL
LIN {X 0,Y 272.998,Z 964.568,A -85,B 0,C 180,E1 -21701.407,E2 -21701.407} C_VEL
LIN {X 0,Y 273.392,Z 961.021,A -85,B 0,C 180,E1 -21706.357,E2 -21706.357} C_VEL
LIN {X 0,Y 275.26,Z 955.619,A -85,B 0,C 180,E1 -21711.748,E2 -21711.748} C_VEL
LIN {X 0,Y 279.247,Z 948.099,A -85,B 0,C 180,E1 -21717.279,E2 -21717.279} C_VEL
LIN {X 0,Y 286.111,Z 938.203,A -85,B 0,C 180,E1 -21723.037,E2 -21723.037} C_VEL
LIN {X 0,Y 295.749,Z 926.427,A -85,B 0,C 180,E1 -21728.468,E2 -21728.468} C_VEL
LIN {X 0,Y 308.63,Z 912.329,A -85,B 0,C 180,E1 -21733.636,E2 -21733.636} C_VEL
LIN {X 0,Y 324.964,Z 895.932,A -85,B 0,C 180,E1 -21738.391,E2 -21738.391} C_VEL
LIN {X 0,Y 342.561,Z 879.263,A -85,B 0,C 180,E1 -21742.196,E2 -21742.196} C_VEL
LIN {X 0,Y 345.779,Z 876.2,A -85,B 0,C 180,E1 -21742.817,E2 -21742.817} C_VEL
LIN {X 0,Y 329.727,Z 887.067,A -85,B 0,C 180,E1 -21746.084,E2 -21746.084} C_VEL
LIN {X 0,Y 316.341,Z 895.907,A -85,B 0,C 180,E1 -21749.62,E2 -21749.62} C_VEL
LIN {X 0,Y 305.348,Z 902.734,A -85,B 0,C 180,E1 -21753.345,E2 -21753.345} C_VEL
LIN {X 0,Y 296.124,Z 907.761,A -85,B 0,C 180,E1 -21757.36,E2 -21757.36} C_VEL
LIN {X 0,Y 288.937,Z 910.728,A -85,B 0,C 180,E1 -21761.435,E2 -21761.435} C_VEL
LIN {X 0,Y 283.548,Z 911.729,A -85,B 0,C 180,E1 -21765.5,E2 -21765.5} C_VEL
LIN {X 0,Y 279.712,Z 910.927,A -85,B 0,C 180,E1 -21769.496,E2 -21769.496} C_VEL
LIN {X 0,Y 277.138,Z 908.494,A -85,B 0,C 180,E1 -21773.37,E2 -21773.37} C_VEL
LIN {X 0,Y 275.432,Z 904.039,A -85,B 0,C 180,E1 -21777.503,E2 -21777.503} C_VEL
LIN {X 0,Y 274.615,Z 897.929,A -85,B 0,C 180,E1 -21781.461,E2 -21781.461} C_VEL
LIN {X 0,Y 274.433,Z 890.313,A -85,B 0,C 180,E1 -21785.226,E2 -21785.226} C_VEL
LIN {X 0,Y 274.82,Z 880.793,A -85,B 0,C 180,E1 -21789.001,E2 -21789.001} C_VEL
LIN {X 0,Y 275.674,Z 870.498,A -85,B 0,C 180,E1 -21792.357,E2 -21792.357} C_VEL
LIN {X 0,Y 277.198,Z 857.439,A -85,B 0,C 180,E1 -21795.911,E2 -21795.911} C_VEL
LIN {X 0,Y 279.257,Z 842.882,A -85,B 0,C 180,E1 -21799.233,E2 -21799.233} C_VEL
LIN {X 0,Y 281.877,Z 826.293,A -85,B 0,C 180,E1 -21802.416,E2 -21802.416} C_VEL
LIN {X 0,Y 284.925,Z 807.951,A -85,B 0,C 180,E1 -21805.349,E2 -21805.349} C_VEL
LIN {X 0,Y 288.304,Z 787.762,A -85,B 0,C 180,E1 -21808.03,E2 -21808.03} C_VEL
LIN {X 0,Y 291.752,Z 766.54,A -85,B 0,C 180,E1 -21810.365,E2 -21810.365} C_VEL
LIN {X 0,Y 294.859,Z 747.2,A -85,B 0,C 180,E1 -21812.168,E2 -21812.168} C_VEL
LIN {X 0,Y 296.39,Z 747.01,A -85,B 0,C 180,E1 -21812.668,E2 -21812.668} C_VEL
LIN {X 0,Y 299.207,Z 744.812,A -85,B 0,C 180,E1 -21813.234,E2 -21813.234} C_VEL
LIN {X 0,Y 303.035,Z 740.398,A -85,B 0,C 180,E1 -21813.747,E2 -21813.747} C_VEL
LIN {X 0,Y 304.712,Z 738.085,A -85,B 0,C 180,E1 -21813.907,E2 -21813.907} C_VEL
LIN {X 0,Y 308.153,Z 735.594,A -85,B 0,C 180,E1 -21814.6,E2 -21814.6} C_VEL
LIN {X 0,Y 312.287,Z 731.048,A -85,B 0,C 180,E1 -21815.193,E2 -21815.193} C_VEL
LIN {X 0,Y 317.192,Z 724.171,A -85,B 0,C 180,E1 -21815.675,E2 -21815.675} C_VEL
LIN {X 0,Y 321.621,Z 719.801,A -85,B 0,C 180,E1 -21816.37,E2 -21816.37} C_VEL
LIN {X 0,Y 326.394,Z 713.32,A -85,B 0,C 180,E1 -21816.901,E2 -21816.901} C_VEL
LIN {X 0,Y 331.706,Z 704.206,A -85,B 0,C 180,E1 -21817.348,E2 -21817.348} C_VEL
LIN {X 0,Y 336.52,Z 698.024,A -85,B 0,C 180,E1 -21817.956,E2 -21817.956} C_VEL
LIN {X 0,Y 341.759,Z 688.852,A -85,B 0,C 180,E1 -21818.442,E2 -21818.442} C_VEL
LIN {X 0,Y 345.773,Z 680.521,A -85,B 0,C 180,E1 -21818.708,E2 -21818.708} C_VEL
LIN {X 0,Y 348.925,Z 676.153,A -85,B 0,C 180,E1 -21819.083,E2 -21819.083} C_VEL
LIN {X 0,Y 344.608,Z 705.687,A -85,B 0,C 180,E1 -21820.39,E2 -21820.39} C_VEL
LIN {X 0,Y 340.76,Z 725.9,A -85,B 0,C 180,E1 -21821.561,E2 -21821.561} C_VEL
LIN {X 0,Y 335.873,Z 746.278,A -85,B 0,C 180,E1 -21823.042,E2 -21823.042} C_VEL
LIN {X 0,Y 330.387,Z 765.45,A -85,B 0,C 180,E1 -21824.769,E2 -21824.769} C_VEL
LIN {X 0,Y 324.254,Z 783.887,A -85,B 0,C 180,E1 -21826.798,E2 -21826.798} C_VEL
LIN {X 0,Y 317.754,Z 801.203,A -85,B 0,C 180,E1 -21829.116,E2 -21829.116} C_VEL
LIN {X 0,Y 311.233,Z 817.009,A -85,B 0,C 180,E1 -21831.68,E2 -21831.68} C_VEL
LIN {X 0,Y 304.434,Z 832.212,A -85,B 0,C 180,E1 -21834.686,E2 -21834.686} C_VEL
LIN {X 0,Y 297.971,Z 845.825,A -85,B 0,C 180,E1 -21837.981,E2 -21837.981} C_VEL
LIN {X 0,Y 292.018,Z 857.892,A -85,B 0,C 180,E1 -21841.579,E2 -21841.579} C_VEL
LIN {X 0,Y 286.751,Z 868.407,A -85,B 0,C 180,E1 -21845.484,E2 -21845.484} C_VEL
LIN {X 0,Y 282.514,Z 876.971,A -85,B 0,C 180,E1 -21849.489,E2 -21849.489} C_VEL
LIN {X 0,Y 279.162,Z 884.043,A -85,B 0,C 180,E1 -21853.777,E2 -21853.777} C_VEL
LIN {X 0,Y 276.738,Z 889.511,A -85,B 0,C 180,E1 -21858.326,E2 -21858.326} C_VEL
LIN {X 0,Y 275.316,Z 893.121,A -85,B 0,C 180,E1 -21862.907,E2 -21862.907} C_VEL
LIN {X 0,Y 274.688,Z 894.887,A -85,B 0,C 180,E1 -21867.288,E2 -21867.288} C_VEL
LIN {X 0,Y 274.606,Z 895.099,A -85,B 0,C 180,E1 -21871.46,E2 -21871.46} C_VEL
LIN {X 0,Y 275.057,Z 893.802,A -85,B 0,C 180,E1 -21875.842,E2 -21875.842} C_VEL
LIN {X 0,Y 276.147,Z 890.921,A -85,B 0,C 180,E1 -21880.22,E2 -21880.22} C_VEL
LIN {X 0,Y 278.099,Z 886.385,A -85,B 0,C 180,E1 -21884.577,E2 -21884.577} C_VEL
LIN {X 0,Y 280.98,Z 880.228,A -85,B 0,C 180,E1 -21888.811,E2 -21888.811} C_VEL
LIN {X 0,Y 284.857,Z 872.344,A -85,B 0,C 180,E1 -21892.931,E2 -21892.931} C_VEL
LIN {X 0,Y 289.699,Z 862.703,A -85,B 0,C 180,E1 -21896.881,E2 -21896.881} C_VEL
LIN {X 0,Y 295.568,Z 850.942,A -85,B 0,C 180,E1 -21900.719,E2 -21900.719} C_VEL
LIN {X 0,Y 301.712,Z 838.27,A -85,B 0,C 180,E1 -21904.061,E2 -21904.061} C_VEL
LIN {X 0,Y 308.232,Z 824.136,A -85,B 0,C 180,E1 -21907.112,E2 -21907.112} C_VEL
LIN {X 0,Y 315.125,Z 808.088,A -85,B 0,C 180,E1 -21909.95,E2 -21909.95} C_VEL
LIN {X 0,Y 321.753,Z 791.181,A -85,B 0,C 180,E1 -21912.404,E2 -21912.404} C_VEL
LIN {X 0,Y 327.984,Z 773.454,A -85,B 0,C 180,E1 -21914.521,E2 -21914.521} C_VEL
LIN {X 0,Y 333.963,Z 753.88,A -85,B 0,C 180,E1 -21916.431,E2 -21916.431} C_VEL
LIN {X 0,Y 339.078,Z 734.096,A -85,B 0,C 180,E1 -21917.997,E2 -21917.997} C_VEL
LIN {X 0,Y 343.327,Z 713.93,A -85,B 0,C 180,E1 -21919.279,E2 -21919.279} C_VEL
LIN {X 0,Y 345.144,Z 703.415,A -85,B 0,C 180,E1 -21919.84,E2 -21919.84} C_VEL
LIN {X 0,Y 345.652,Z 696.184,A -85,B 0,C 180,E1 -21920.307,E2 -21920.307} C_VEL
LIN {X 0,Y 344.547,Z 678.435,A -85,B 0,C 180,E1 -21921.869,E2 -21921.869} C_VEL
LIN {X 0,Y 345.016,Z 671.141,A -85,B 0,C 180,E1 -21922.293,E2 -21922.293} C_VEL
LIN {X 0,Y 351.317,Z 629.328,A -85,B 0,C 180,E1 -21923.731,E2 -21923.731} C_VEL
LIN {X 0,Y 358.541,Z 578.263,A -85,B 0,C 180,E1 -21925.122,E2 -21925.122} C_VEL
LIN {X 0,Y 364.196,Z 528.171,A -85,B 0,C 180,E1 -21926.252,E2 -21926.252} C_VEL
LIN {X 0,Y 369.295,Z 466.763,A -85,B 0,C 180,E1 -21927.403,E2 -21927.403} C_VEL
LIN {X 0,Y 371.189,Z 444.83,A -85,B 0,C 180,E1 -21927.807,E2 -21927.807} C_VEL
LIN {X 0,Y 377.281,Z 418.51,A -85,B 0,C 180,E1 -21928.66,E2 -21928.66} C_VEL
LIN {X 0,Y 372.706,Z 403.689,A -85,B 0,C 180,E1 -21931.65,E2 -21931.65} C_VEL
LIN {X 0,Y 368.179,Z 390.746,A -85,B 0,C 180,E1 -21934.723,E2 -21934.723} C_VEL
LIN {X 0,Y 364.132,Z 380.11,A -85,B 0,C 180,E1 -21937.732,E2 -21937.732} C_VEL
LIN {X 0,Y 360.372,Z 371.096,A -85,B 0,C 180,E1 -21940.72,E2 -21940.72} C_VEL
LIN {X 0,Y 357.05,Z 363.402,A -85,B 0,C 180,E1 -21943.821,E2 -21943.821} C_VEL
LIN {X 0,Y 354.771,Z 358.473,A -85,B 0,C 180,E1 -21946.222,E2 -21946.222} C_VEL
LIN {X 0,Y 353.222,Z 354.758,A -85,B 0,C 180,E1 -21948.323,E2 -21948.323} C_VEL
LIN {X 0,Y 351.316,Z 350.5,A -85,B 0,C 180,E1 -21951.159,E2 -21951.159} C_VEL
LIN {X 0,Y 349.637,Z 346.785,A -85,B 0,C 180,E1 -21954.667,E2 -21954.667} C_VEL
LIN {X 0,Y 349.523,Z 345.779,A -85,B 0,C 180,E1 -21955.57,E2 -21955.57} C_VEL
LIN {X 0,Y 348.875,Z 344.313,A -85,B 0,C 180,E1 -21961.807,E2 -21961.807} C_VEL
LIN {X 0,Y 350.785,Z 345.628,A -85,B 0,C 180,E1 -21966.876,E2 -21966.876} C_VEL
LIN {X 0,Y 351.232,Z 346.212,A -85,B 0,C 180,E1 -21967.648,E2 -21967.648} C_VEL
LIN {X 0,Y 352.621,Z 357.497,A -85,B 0,C 180,E1 -21971.532,E2 -21971.532} C_VEL
LIN {X 0,Y 355.325,Z 369.691,A -85,B 0,C 180,E1 -21975.213,E2 -21975.213} C_VEL
LIN {X 0,Y 360.791,Z 388.654,A -85,B 0,C 180,E1 -21980.05,E2 -21980.05} C_VEL
LIN {X 0,Y 363.902,Z 398.437,A -85,B 0,C 180,E1 -21982.198,E2 -21982.198} C_VEL
LIN {X 0,Y 368.896,Z 415.425,A -85,B 0,C 180,E1 -21985.248,E2 -21985.248} C_VEL
LIN {X 0,Y 347.702,Z 578.804,A -85,B 0,C 180,E1 -21989.614,E2 -21989.614} C_VEL
LIN {X 0,Y 343.26,Z 640.84,A -85,B 0,C 180,E1 -21990.923,E2 -21990.923} C_VEL
LIN {X 0,Y 339.632,Z 674.063,A -85,B 0,C 180,E1 -21991.823,E2 -21991.823} C_VEL
LIN {X 0,Y 334.92,Z 706.612,A -85,B 0,C 180,E1 -21992.931,E2 -21992.931} C_VEL
LIN {X 0,Y 329.773,Z 736.672,A -85,B 0,C 180,E1 -21994.209,E2 -21994.209} C_VEL
LIN {X 0,Y 324.267,Z 764.925,A -85,B 0,C 180,E1 -21995.734,E2 -21995.734} C_VEL
LIN {X 0,Y 318.05,Z 793.74,A -85,B 0,C 180,E1 -21997.605,E2 -21997.605} C_VEL
LIN {X 0,Y 313.326,Z 813.545,A -85,B 0,C 180,E1 -21999.153,E2 -21999.153} C_VEL
LIN {X 0,Y 308.022,Z 832.534,A -85,B 0,C 180,E1 -22000.998,E2 -22000.998} C_VEL
LIN {X 0,Y 302.499,Z 849.927,A -85,B 0,C 180,E1 -22003.072,E2 -22003.072} C_VEL
LIN {X 0,Y 296.599,Z 866.61,A -85,B 0,C 180,E1 -22005.476,E2 -22005.476} C_VEL
LIN {X 0,Y 290.406,Z 882.917,A -85,B 0,C 180,E1 -22008.355,E2 -22008.355} C_VEL
LIN {X 0,Y 284.535,Z 897.684,A -85,B 0,C 180,E1 -22011.538,E2 -22011.538} C_VEL
LIN {X 0,Y 278.87,Z 911.797,A -85,B 0,C 180,E1 -22015.243,E2 -22015.243} C_VEL
LIN {X 0,Y 274.014,Z 924.334,A -85,B 0,C 180,E1 -22019.279,E2 -22019.279} C_VEL
LIN {X 0,Y 270.15,Z 935.188,A -85,B 0,C 180,E1 -22023.631,E2 -22023.631} C_VEL
LIN {X 0,Y 267.426,Z 944.444,A -85,B 0,C 180,E1 -22028.275,E2 -22028.275} C_VEL
LIN {X 0,Y 265.952,Z 951.758,A -85,B 0,C 180,E1 -22032.947,E2 -22032.947} C_VEL
LIN {X 0,Y 265.54,Z 957.219,A -85,B 0,C 180,E1 -22037.606,E2 -22037.606} C_VEL
LIN {X 0,Y 265.804,Z 960.804,A -85,B 0,C 180,E1 -22041.999,E2 -22041.999} C_VEL
LIN {X 0,Y 266.299,Z 962.817,A -85,B 0,C 180,E1 -22046.125,E2 -22046.125} C_VEL
LIN {X 0,Y 266.367,Z 964.649,A -85,B 0,C 180,E1 -22050,E2 -22050} C_VEL
LIN {X 0,Y 266.018,Z 965.374,A -85,B 0,C 180,E1 -22053.448,E2 -22053.448} C_VEL
LIN {X 0,Y 265.461,Z 965.112,A -85,B 0,C 180,E1 -22057.14,E2 -22057.14} C_VEL
LIN {X 0,Y 265.046,Z 963.601,A -85,B 0,C 180,E1 -22061.534,E2 -22061.534} C_VEL
LIN {X 0,Y 265.547,Z 959.968,A -85,B 0,C 180,E1 -22067.08,E2 -22067.08} C_VEL
LIN {X 0,Y 267.446,Z 955.13,A -85,B 0,C 180,E1 -22072.186,E2 -22072.186} C_VEL
LIN {X 0,Y 272.085,Z 947.409,A -85,B 0,C 180,E1 -22078.299,E2 -22078.299} C_VEL
LIN {X 0,Y 279.501,Z 937.848,A -85,B 0,C 180,E1 -22084.17,E2 -22084.17} C_VEL
LIN {X 0,Y 289.909,Z 926.294,A -85,B 0,C 180,E1 -22089.725,E2 -22089.725} C_VEL
LIN {X 0,Y 304.431,Z 911.944,A -85,B 0,C 180,E1 -22095.19,E2 -22095.19} C_VEL
LIN {X 0,Y 321.084,Z 896.78,A -85,B 0,C 180,E1 -22099.726,E2 -22099.726} C_VEL
LIN {X 0,Y 335.98,Z 883.69,A -85,B 0,C 180,E1 -22102.887,E2 -22102.887} C_VEL
LIN {X 0,Y 320.197,Z 893.303,A -85,B 0,C 180,E1 -22106.231,E2 -22106.231} C_VEL
LIN {X 0,Y 306.371,Z 901.354,A -85,B 0,C 180,E1 -22110.044,E2 -22110.044} C_VEL
LIN {X 0,Y 295.108,Z 907.303,A -85,B 0,C 180,E1 -22114.082,E2 -22114.082} C_VEL
LIN {X 0,Y 286.494,Z 911.032,A -85,B 0,C 180,E1 -22118.072,E2 -22118.072} C_VEL
LIN {X 0,Y 279.523,Z 912.961,A -85,B 0,C 180,E1 -22122.299,E2 -22122.299} C_VEL
LIN {X 0,Y 274.597,Z 913.028,A -85,B 0,C 180,E1 -22126.309,E2 -22126.309} C_VEL
LIN {X 0,Y 270.967,Z 911.374,A -85,B 0,C 180,E1 -22130.442,E2 -22130.442} C_VEL
LIN {X 0,Y 268.494,Z 907.861,A -85,B 0,C 180,E1 -22134.658,E2 -22134.658} C_VEL
LIN {X 0,Y 267.113,Z 902.722,A -85,B 0,C 180,E1 -22138.713,E2 -22138.713} C_VEL
LIN {X 0,Y 266.496,Z 895.934,A -85,B 0,C 180,E1 -22142.695,E2 -22142.695} C_VEL
LIN {X 0,Y 266.5,Z 887.774,A -85,B 0,C 180,E1 -22146.463,E2 -22146.463} C_VEL
LIN {X 0,Y 267.095,Z 877.385,A -85,B 0,C 180,E1 -22150.352,E2 -22150.352} C_VEL
LIN {X 0,Y 268.276,Z 865.508,A -85,B 0,C 180,E1 -22154.02,E2 -22154.02} C_VEL
LIN {X 0,Y 270.015,Z 852.195,A -85,B 0,C 180,E1 -22157.455,E2 -22157.455} C_VEL
LIN {X 0,Y 272.488,Z 835.962,A -85,B 0,C 180,E1 -22160.964,E2 -22160.964} C_VEL
LIN {X 0,Y 275.487,Z 817.977,A -85,B 0,C 180,E1 -22164.214,E2 -22164.214} C_VEL
LIN {X 0,Y 278.801,Z 798.85,A -85,B 0,C 180,E1 -22167.096,E2 -22167.096} C_VEL
LIN {X 0,Y 282.236,Z 778.557,A -85,B 0,C 180,E1 -22169.618,E2 -22169.618} C_VEL
LIN {X 0,Y 285.146,Z 761.379,A -85,B 0,C 180,E1 -22171.457,E2 -22171.457} C_VEL
LIN {X 0,Y 286.729,Z 761.147,A -85,B 0,C 180,E1 -22172.01,E2 -22172.01} C_VEL
LIN {X 0,Y 289.74,Z 758.909,A -85,B 0,C 180,E1 -22172.643,E2 -22172.643} C_VEL
LIN {X 0,Y 294.315,Z 754.082,A -85,B 0,C 180,E1 -22173.276,E2 -22173.276} C_VEL
LIN {X 0,Y 297.283,Z 752.301,A -85,B 0,C 180,E1 -22173.941,E2 -22173.941} C_VEL
LIN {X 0,Y 301.725,Z 748.238,A -85,B 0,C 180,E1 -22174.635,E2 -22174.635} C_VEL
LIN {X 0,Y 305.43,Z 743.832,A -85,B 0,C 180,E1 -22175.056,E2 -22175.056} C_VEL
LIN {X 0,Y 309.582,Z 740.494,A -85,B 0,C 180,E1 -22175.775,E2 -22175.775} C_VEL
LIN {X 0,Y 314.388,Z 735.324,A -85,B 0,C 180,E1 -22176.37,E2 -22176.37} C_VEL
LIN {X 0,Y 318.866,Z 729.325,A -85,B 0,C 180,E1 -22176.794,E2 -22176.794} C_VEL
LIN {X 0,Y 324.23,Z 723.906,A -85,B 0,C 180,E1 -22177.522,E2 -22177.522} C_VEL
LIN {X 0,Y 329.942,Z 716.128,A -85,B 0,C 180,E1 -22178.077,E2 -22178.077} C_VEL
LIN {X 0,Y 334.161,Z 709.076,A -85,B 0,C 180,E1 -22178.375,E2 -22178.375} C_VEL
LIN {X 0,Y 339.511,Z 702.211,A -85,B 0,C 180,E1 -22178.996,E2 -22178.996} C_VEL
LIN {X 0,Y 340.39,Z 701.1,A -85,B 0,C 180,E1 -22179.098,E2 -22179.098} C_VEL
LIN {X 0,Y 336.602,Z 721.861,A -85,B 0,C 180,E1 -22180.232,E2 -22180.232} C_VEL
LIN {X 0,Y 331.63,Z 743.031,A -85,B 0,C 180,E1 -22181.698,E2 -22181.698} C_VEL
LIN {X 0,Y 326.08,Z 762.53,A -85,B 0,C 180,E1 -22183.386,E2 -22183.386} C_VEL
LIN {X 0,Y 319.86,Z 781.204,A -85,B 0,C 180,E1 -22185.371,E2 -22185.371} C_VEL
LIN {X 0,Y 313.009,Z 799.27,A -85,B 0,C 180,E1 -22187.721,E2 -22187.721} C_VEL
LIN {X 0,Y 305.9,Z 816.106,A -85,B 0,C 180,E1 -22190.402,E2 -22190.402} C_VEL
LIN {X 0,Y 298.762,Z 831.616,A -85,B 0,C 180,E1 -22193.435,E2 -22193.435} C_VEL
LIN {X 0,Y 291.947,Z 845.488,A -85,B 0,C 180,E1 -22196.771,E2 -22196.771} C_VEL
LIN {X 0,Y 285.632,Z 857.785,A -85,B 0,C 180,E1 -22200.423,E2 -22200.423} C_VEL
LIN {X 0,Y 280.009,Z 868.505,A -85,B 0,C 180,E1 -22204.4,E2 -22204.4} C_VEL
LIN {X 0,Y 275.246,Z 877.627,A -85,B 0,C 180,E1 -22208.699,E2 -22208.699} C_VEL
LIN {X 0,Y 271.595,Z 884.884,A -85,B 0,C 180,E1 -22213.178,E2 -22213.178} C_VEL
LIN {X 0,Y 268.992,Z 890.399,A -85,B 0,C 180,E1 -22217.856,E2 -22217.856} C_VEL
LIN {X 0,Y 267.473,Z 893.986,A -85,B 0,C 180,E1 -22222.482,E2 -22222.482} C_VEL
LIN {X 0,Y 266.772,Z 895.828,A -85,B 0,C 180,E1 -22226.992,E2 -22226.992} C_VEL
LIN {X 0,Y 266.662,Z 896.121,A -85,B 0,C 180,E1 -22231.289,E2 -22231.289} C_VEL
LIN {X 0,Y 267.113,Z 894.908,A -85,B 0,C 180,E1 -22235.801,E2 -22235.801} C_VEL
LIN {X 0,Y 268.239,Z 892.115,A -85,B 0,C 180,E1 -22240.307,E2 -22240.307} C_VEL
LIN {X 0,Y 270.266,Z 887.671,A -85,B 0,C 180,E1 -22244.79,E2 -22244.79} C_VEL
LIN {X 0,Y 273.328,Z 881.472,A -85,B 0,C 180,E1 -22249.222,E2 -22249.222} C_VEL
LIN {X 0,Y 277.515,Z 873.376,A -85,B 0,C 180,E1 -22253.574,E2 -22253.574} C_VEL
LIN {X 0,Y 282.598,Z 863.747,A -85,B 0,C 180,E1 -22257.613,E2 -22257.613} C_VEL
LIN {X 0,Y 288.734,Z 851.984,A -85,B 0,C 180,E1 -22261.528,E2 -22261.528} C_VEL
LIN {X 0,Y 295.141,Z 839.32,A -85,B 0,C 180,E1 -22264.929,E2 -22264.929} C_VEL
LIN {X 0,Y 301.919,Z 825.203,A -85,B 0,C 180,E1 -22268.024,E2 -22268.024} C_VEL
LIN {X 0,Y 308.9,Z 809.554,A -85,B 0,C 180,E1 -22270.833,E2 -22270.833} C_VEL
LIN {X 0,Y 315.928,Z 792.228,A -85,B 0,C 180,E1 -22273.376,E2 -22273.376} C_VEL
LIN {X 0,Y 322.368,Z 774.489,A -85,B 0,C 180,E1 -22275.511,E2 -22275.511} C_VEL
LIN {X 0,Y 328.282,Z 755.819,A -85,B 0,C 180,E1 -22277.355,E2 -22277.355} C_VEL
LIN {X 0,Y 333.552,Z 736.201,A -85,B 0,C 180,E1 -22278.931,E2 -22278.931} C_VEL
LIN {X 0,Y 338.068,Z 715.486,A -85,B 0,C 180,E1 -22280.263,E2 -22280.263} C_VEL
LIN {X 0,Y 341.601,Z 694.386,A -85,B 0,C 180,E1 -22281.325,E2 -22281.325} C_VEL
LIN {X 0,Y 345.016,Z 671.141,A -85,B 0,C 180,E1 -22282.293,E2 -22282.293} C_VEL
LIN {X 0,Y 345.559,Z 663.804,A -85,B 0,C 180,E1 -22282.709,E2 -22282.709} C_VEL
LIN {X 0,Y 344.886,Z 645.737,A -85,B 0,C 180,E1 -22284.174,E2 -22284.174} C_VEL
LIN {X 0,Y 345.461,Z 638.348,A -85,B 0,C 180,E1 -22284.547,E2 -22284.547} C_VEL
LIN {X 0,Y 352.686,Z 589.505,A -85,B 0,C 180,E1 -22285.92,E2 -22285.92} C_VEL
LIN {X 0,Y 358.626,Z 541.142,A -85,B 0,C 180,E1 -22287.058,E2 -22287.058} C_VEL
LIN {X 0,Y 363.158,Z 492.249,A -85,B 0,C 180,E1 -22288.02,E2 -22288.02} C_VEL
LIN {X 0,Y 366.865,Z 447.449,A -85,B 0,C 180,E1 -22288.828,E2 -22288.828} C_VEL
LIN {X 0,Y 372.743,Z 422.289,A -85,B 0,C 180,E1 -22289.625,E2 -22289.625} C_VEL
LIN {X 0,Y 368.415,Z 408.009,A -85,B 0,C 180,E1 -22292.611,E2 -22292.611} C_VEL
LIN {X 0,Y 364.236,Z 395.66,A -85,B 0,C 180,E1 -22295.64,E2 -22295.64} C_VEL
LIN {X 0,Y 360.156,Z 384.746,A -85,B 0,C 180,E1 -22298.843,E2 -22298.843} C_VEL
LIN {X 0,Y 356.22,Z 374.962,A -85,B 0,C 180,E1 -22302.311,E2 -22302.311} C_VEL
LIN {X 0,Y 352.759,Z 366.756,A -85,B 0,C 180,E1 -22305.975,E2 -22305.975} C_VEL
LIN {X 0,Y 350.734,Z 362.044,A -85,B 0,C 180,E1 -22308.722,E2 -22308.722} C_VEL
LIN {X 0,Y 349.13,Z 358.063,A -85,B 0,C 180,E1 -22311.435,E2 -22311.435} C_VEL
LIN {X 0,Y 347.607,Z 354.308,A -85,B 0,C 180,E1 -22314.967,E2 -22314.967} C_VEL
LIN {X 0,Y 347.482,Z 353.459,A -85,B 0,C 180,E1 -22315.875,E2 -22315.875} C_VEL
LIN {X 0,Y 347.085,Z 352.111,A -85,B 0,C 180,E1 -22321.816,E2 -22321.816} C_VEL
LIN {X 0,Y 349.109,Z 353.469,A -85,B 0,C 180,E1 -22326.909,E2 -22326.909} C_VEL
LIN {X 0,Y 349.322,Z 353.983,A -85,B 0,C 180,E1 -22327.359,E2 -22327.359} C_VEL
LIN {X 0,Y 350.507,Z 364.551,A -85,B 0,C 180,E1 -22331.019,E2 -22331.019} C_VEL
LIN {X 0,Y 352.914,Z 376.48,A -85,B 0,C 180,E1 -22334.647,E2 -22334.647} C_VEL
LIN {X 0,Y 358.177,Z 395.672,A -85,B 0,C 180,E1 -22339.572,E2 -22339.572} C_VEL
LIN {X 0,Y 361.075,Z 404.965,A -85,B 0,C 180,E1 -22341.611,E2 -22341.611} C_VEL
LIN {X 0,Y 364.975,Z 419.19,A -85,B 0,C 180,E1 -22344.206,E2 -22344.206} C_VEL
LIN {X 0,Y 343.906,Z 575.914,A -85,B 0,C 180,E1 -22348.395,E2 -22348.395} C_VEL
LIN {X 0,Y 339.36,Z 637.568,A -85,B 0,C 180,E1 -22349.7,E2 -22349.7} C_VEL
LIN {X 0,Y 335.582,Z 671.204,A -85,B 0,C 180,E1 -22350.6,E2 -22350.6} C_VEL
LIN {X 0,Y 330.752,Z 703.669,A -85,B 0,C 180,E1 -22351.69,E2 -22351.69} C_VEL
LIN {X 0,Y 325.385,Z 734.286,A -85,B 0,C 180,E1 -22352.975,E2 -22352.975} C_VEL
LIN {X 0,Y 319.944,Z 761.293,A -85,B 0,C 180,E1 -22354.406,E2 -22354.406} C_VEL
LIN {X 0,Y 313.887,Z 788.844,A -85,B 0,C 180,E1 -22356.145,E2 -22356.145} C_VEL
LIN {X 0,Y 308.688,Z 810.28,A -85,B 0,C 180,E1 -22357.781,E2 -22357.781} C_VEL
LIN {X 0,Y 303.137,Z 829.589,A -85,B 0,C 180,E1 -22359.629,E2 -22359.629} C_VEL
LIN {X 0,Y 297.3,Z 847.226,A -85,B 0,C 180,E1 -22361.7,E2 -22361.7} C_VEL
LIN {X 0,Y 290.87,Z 864.744,A -85,B 0,C 180,E1 -22364.214,E2 -22364.214} C_VEL
LIN {X 0,Y 284.444,Z 880.988,A -85,B 0,C 180,E1 -22367.089,E2 -22367.089} C_VEL
LIN {X 0,Y 278.335,Z 895.629,A -85,B 0,C 180,E1 -22370.25,E2 -22370.25} C_VEL
LIN {X 0,Y 272.276,Z 909.882,A -85,B 0,C 180,E1 -22374.015,E2 -22374.015} C_VEL
LIN {X 0,Y 267.294,Z 921.921,A -85,B 0,C 180,E1 -22377.914,E2 -22377.914} C_VEL
LIN {X 0,Y 263.198,Z 932.582,A -85,B 0,C 180,E1 -22382.142,E2 -22382.142} C_VEL
LIN {X 0,Y 260.13,Z 941.834,A -85,B 0,C 180,E1 -22386.733,E2 -22386.733} C_VEL
LIN {X 0,Y 258.224,Z 949.726,A -85,B 0,C 180,E1 -22391.721,E2 -22391.721} C_VEL
LIN {X 0,Y 257.569,Z 955.485,A -85,B 0,C 180,E1 -22396.531,E2 -22396.531} C_VEL
LIN {X 0,Y 257.778,Z 959.51,A -85,B 0,C 180,E1 -22401.299,E2 -22401.299} C_VEL
LIN {X 0,Y 258.287,Z 961.671,A -85,B 0,C 180,E1 -22405.56,E2 -22405.56} C_VEL
LIN {X 0,Y 258.519,Z 962.811,A -85,B 0,C 180,E1 -22408.892,E2 -22408.892} C_VEL
LIN {X 0,Y 258.193,Z 964.018,A -85,B 0,C 180,E1 -22412.886,E2 -22412.886} C_VEL
LIN {X 0,Y 257.543,Z 963.94,A -85,B 0,C 180,E1 -22417.137,E2 -22417.137} C_VEL
LIN {X 0,Y 257.104,Z 962.669,A -85,B 0,C 180,E1 -22421.466,E2 -22421.466} C_VEL
LIN {X 0,Y 257.44,Z 959.909,A -85,B 0,C 180,E1 -22426.471,E2 -22426.471} C_VEL
LIN {X 0,Y 259.646,Z 954.661,A -85,B 0,C 180,E1 -22432.65,E2 -22432.65} C_VEL
LIN {X 0,Y 264.211,Z 947.807,A -85,B 0,C 180,E1 -22438.599,E2 -22438.599} C_VEL
LIN {X 0,Y 272.006,Z 938.514,A -85,B 0,C 180,E1 -22444.735,E2 -22444.735} C_VEL
LIN {X 0,Y 283.522,Z 926.959,A -85,B 0,C 180,E1 -22450.726,E2 -22450.726} C_VEL
LIN {X 0,Y 298.295,Z 913.641,A -85,B 0,C 180,E1 -22456.111,E2 -22456.111} C_VEL
LIN {X 0,Y 315.481,Z 899.188,A -85,B 0,C 180,E1 -22460.663,E2 -22460.663} C_VEL
LIN {X 0,Y 326.168,Z 890.562,A -85,B 0,C 180,E1 -22462.948,E2 -22462.948} C_VEL
LIN {X 0,Y 310.014,Z 899.337,A -85,B 0,C 180,E1 -22466.528,E2 -22466.528} C_VEL
LIN {X 0,Y 296.356,Z 906.225,A -85,B 0,C 180,E1 -22470.488,E2 -22470.488} C_VEL
LIN {X 0,Y 285.264,Z 911.069,A -85,B 0,C 180,E1 -22474.683,E2 -22474.683} C_VEL
LIN {X 0,Y 276.501,Z 913.864,A -85,B 0,C 180,E1 -22479.022,E2 -22479.022} C_VEL
LIN {X 0,Y 269.849,Z 914.678,A -85,B 0,C 180,E1 -22483.422,E2 -22483.422} C_VEL
LIN {X 0,Y 265.25,Z 913.719,A -85,B 0,C 180,E1 -22487.592,E2 -22487.592} C_VEL
LIN {X 0,Y 261.959,Z 911.019,A -85,B 0,C 180,E1 -22491.881,E2 -22491.881} C_VEL
LIN {X 0,Y 259.841,Z 906.46,A -85,B 0,C 180,E1 -22496.249,E2 -22496.249} C_VEL
LIN {X 0,Y 258.767,Z 900.288,A -85,B 0,C 180,E1 -22500.443,E2 -22500.443} C_VEL
LIN {X 0,Y 258.435,Z 892.664,A -85,B 0,C 180,E1 -22504.438,E2 -22504.438} C_VEL
LIN {X 0,Y 258.727,Z 883.15,A -85,B 0,C 180,E1 -22508.445,E2 -22508.445} C_VEL
LIN {X 0,Y 259.6,Z 872.174,A -85,B 0,C 180,E1 -22512.23,E2 -22512.23} C_VEL
LIN {X 0,Y 261.198,Z 858.773,A -85,B 0,C 180,E1 -22516.084,E2 -22516.084} C_VEL
LIN {X 0,Y 263.291,Z 844.477,A -85,B 0,C 180,E1 -22519.524,E2 -22519.524} C_VEL
LIN {X 0,Y 266.029,Z 827.779,A -85,B 0,C 180,E1 -22522.893,E2 -22522.893} C_VEL
LIN {X 0,Y 269.345,Z 808.814,A -85,B 0,C 180,E1 -22526.098,E2 -22526.098} C_VEL
LIN {X 0,Y 272.919,Z 788.641,A -85,B 0,C 180,E1 -22528.921,E2 -22528.921} C_VEL
LIN {X 0,Y 275.484,Z 774.071,A -85,B 0,C 180,E1 -22530.691,E2 -22530.691} C_VEL
LIN {X 0,Y 277.117,Z 773.825,A -85,B 0,C 180,E1 -22531.304,E2 -22531.304} C_VEL
LIN {X 0,Y 279.822,Z 772.019,A -85,B 0,C 180,E1 -22531.928,E2 -22531.928} C_VEL
LIN {X 0,Y 283.993,Z 768.125,A -85,B 0,C 180,E1 -22532.595,E2 -22532.595} C_VEL
LIN {X 0,Y 287.484,Z 766.13,A -85,B 0,C 180,E1 -22533.411,E2 -22533.411} C_VEL
LIN {X 0,Y 292.129,Z 762.099,A -85,B 0,C 180,E1 -22534.148,E2 -22534.148} C_VEL
LIN {X 0,Y 293.991,Z 760.179,A -85,B 0,C 180,E1 -22534.373,E2 -22534.373} C_VEL
LIN {X 0,Y 298.345,Z 757.201,A -85,B 0,C 180,E1 -22535.202,E2 -22535.202} C_VEL
LIN {X 0,Y 303.846,Z 751.934,A -85,B 0,C 180,E1 -22535.949,E2 -22535.949} C_VEL
LIN {X 0,Y 306.307,Z 749.242,A -85,B 0,C 180,E1 -22536.217,E2 -22536.217} C_VEL
LIN {X 0,Y 311.901,Z 744.537,A -85,B 0,C 180,E1 -22537.037,E2 -22537.037} C_VEL
LIN {X 0,Y 317.585,Z 738.191,A -85,B 0,C 180,E1 -22537.647,E2 -22537.647} C_VEL
LIN {X 0,Y 320.622,Z 734.323,A -85,B 0,C 180,E1 -22537.906,E2 -22537.906} C_VEL
LIN {X 0,Y 326.669,Z 728.199,A -85,B 0,C 180,E1 -22538.64,E2 -22538.64} C_VEL
LIN {X 0,Y 331.79,Z 721.533,A -85,B 0,C 180,E1 -22539.1,E2 -22539.1} C_VEL
LIN {X 0,Y 327.148,Z 741.267,A -85,B 0,C 180,E1 -22540.444,E2 -22540.444} C_VEL
LIN {X 0,Y 321.749,Z 760.218,A -85,B 0,C 180,E1 -22542.035,E2 -22542.035} C_VEL
LIN {X 0,Y 315.427,Z 779.078,A -85,B 0,C 180,E1 -22543.98,E2 -22543.98} C_VEL
LIN {X 0,Y 308.575,Z 796.943,A -85,B 0,C 180,E1 -22546.239,E2 -22546.239} C_VEL
LIN {X 0,Y 301.421,Z 813.63,A -85,B 0,C 180,E1 -22548.816,E2 -22548.816} C_VEL
LIN {X 0,Y 294.083,Z 829.245,A -85,B 0,C 180,E1 -22551.771,E2 -22551.771} C_VEL
LIN {X 0,Y 287.194,Z 842.907,A -85,B 0,C 180,E1 -22554.938,E2 -22554.938} C_VEL
LIN {X 0,Y 280.689,Z 855.168,A -85,B 0,C 180,E1 -22558.422,E2 -22558.422} C_VEL
LIN {X 0,Y 274.762,Z 866.016,A -85,B 0,C 180,E1 -22562.237,E2 -22562.237} C_VEL
LIN {X 0,Y 269.581,Z 875.414,A -85,B 0,C 180,E1 -22566.386,E2 -22566.386} C_VEL
LIN {X 0,Y 265.321,Z 883.278,A -85,B 0,C 180,E1 -22570.86,E2 -22570.86} C_VEL
LIN {X 0,Y 262.232,Z 889.286,A -85,B 0,C 180,E1 -22575.424,E2 -22575.424} C_VEL
LIN {X 0,Y 260.213,Z 893.564,A -85,B 0,C 180,E1 -22580.042,E2 -22580.042} C_VEL
LIN {X 0,Y 259.111,Z 896.158,A -85,B 0,C 180,E1 -22584.686,E2 -22584.686} C_VEL
LIN {X 0,Y 258.716,Z 897.151,A -85,B 0,C 180,E1 -22589.114,E2 -22589.114} C_VEL
LIN {X 0,Y 258.893,Z 896.681,A -85,B 0,C 180,E1 -22593.764,E2 -22593.764} C_VEL
LIN {X 0,Y 259.735,Z 894.645,A -85,B 0,C 180,E1 -22598.412,E2 -22598.412} C_VEL
LIN {X 0,Y 261.405,Z 891.002,A -85,B 0,C 180,E1 -22603.043,E2 -22603.043} C_VEL
LIN {X 0,Y 264.12,Z 885.658,A -85,B 0,C 180,E1 -22607.629,E2 -22607.629} C_VEL
LIN {X 0,Y 267.957,Z 878.492,A -85,B 0,C 180,E1 -22612.141,E2 -22612.141} C_VEL
LIN {X 0,Y 272.742,Z 869.847,A -85,B 0,C 180,E1 -22616.333,E2 -22616.333} C_VEL
LIN {X 0,Y 278.618,Z 859.197,A -85,B 0,C 180,E1 -22620.399,E2 -22620.399} C_VEL
LIN {X 0,Y 285.198,Z 846.976,A -85,B 0,C 180,E1 -22624.122,E2 -22624.122} C_VEL
LIN {X 0,Y 292.279,Z 833.18,A -85,B 0,C 180,E1 -22627.513,E2 -22627.513} C_VEL
LIN {X 0,Y 299.457,Z 818.252,A -85,B 0,C 180,E1 -22630.499,E2 -22630.499} C_VEL
LIN {X 0,Y 306.505,Z 802.316,A -85,B 0,C 180,E1 -22633.113,E2 -22633.113} C_VEL
LIN {X 0,Y 313.469,Z 784.852,A -85,B 0,C 180,E1 -22635.459,E2 -22635.459} C_VEL
LIN {X 0,Y 319.752,Z 767.032,A -85,B 0,C 180,E1 -22637.428,E2 -22637.428} C_VEL
LIN {X 0,Y 325.624,Z 747.606,A -85,B 0,C 180,E1 -22639.18,E2 -22639.18} C_VEL
LIN {X 0,Y 330.583,Z 728.05,A -85,B 0,C 180,E1 -22640.605,E2 -22640.605} C_VEL
LIN {X 0,Y 334.804,Z 706.92,A -85,B 0,C 180,E1 -22641.83,E2 -22641.83} C_VEL
LIN {X 0,Y 340.845,Z 668.017,A -85,B 0,C 180,E1 -22643.512,E2 -22643.512} C_VEL
LIN {X 0,Y 345.461,Z 638.348,A -85,B 0,C 180,E1 -22644.547,E2 -22644.547} C_VEL
LIN {X 0,Y 346.093,Z 630.92,A -85,B 0,C 180,E1 -22644.908,E2 -22644.908} C_VEL
LIN {X 0,Y 345.73,Z 611.532,A -85,B 0,C 180,E1 -22646.344,E2 -22646.344} C_VEL
LIN {X 0,Y 346.295,Z 605.133,A -85,B 0,C 180,E1 -22646.631,E2 -22646.631} C_VEL
LIN {X 0,Y 352.764,Z 556.34,A -85,B 0,C 180,E1 -22647.83,E2 -22647.83} C_VEL
LIN {X 0,Y 357.731,Z 508.112,A -85,B 0,C 180,E1 -22648.822,E2 -22648.822} C_VEL
LIN {X 0,Y 362.648,Z 450.247,A -85,B 0,C 180,E1 -22649.871,E2 -22649.871} C_VEL
LIN {X 0,Y 368.302,Z 426.072,A -85,B 0,C 180,E1 -22650.63,E2 -22650.63} C_VEL
LIN {X 0,Y 364.176,Z 412.156,A -85,B 0,C 180,E1 -22653.634,E2 -22653.634} C_VEL
LIN {X 0,Y 360.093,Z 399.779,A -85,B 0,C 180,E1 -22656.821,E2 -22656.821} C_VEL
LIN {X 0,Y 356.102,Z 388.919,A -85,B 0,C 180,E1 -22660.181,E2 -22660.181} C_VEL
LIN {X 0,Y 352.793,Z 380.573,A -85,B 0,C 180,E1 -22663.366,E2 -22663.366} C_VEL
LIN {X 0,Y 350.053,Z 373.712,A -85,B 0,C 180,E1 -22666.538,E2 -22666.538} C_VEL
LIN {X 0,Y 348.405,Z 369.611,A -85,B 0,C 180,E1 -22668.914,E2 -22668.914} C_VEL
LIN {X 0,Y 346.952,Z 365.624,A -85,B 0,C 180,E1 -22671.715,E2 -22671.715} C_VEL
LIN {X 0,Y 345.586,Z 361.831,A -85,B 0,C 180,E1 -22675.27,E2 -22675.27} C_VEL
LIN {X 0,Y 345.451,Z 361.14,A -85,B 0,C 180,E1 -22676.183,E2 -22676.183} C_VEL
LIN {X 0,Y 345.294,Z 359.908,A -85,B 0,C 180,E1 -22681.825,E2 -22681.825} C_VEL
LIN {X 0,Y 347.292,Z 361.192,A -85,B 0,C 180,E1 -22686.641,E2 -22686.641} C_VEL
LIN {X 0,Y 347.467,Z 361.736,A -85,B 0,C 180,E1 -22687.066,E2 -22687.066} C_VEL
LIN {X 0,Y 348.421,Z 371.605,A -85,B 0,C 180,E1 -22690.5,E2 -22690.5} C_VEL
LIN {X 0,Y 350.524,Z 383.357,A -85,B 0,C 180,E1 -22694.101,E2 -22694.101} C_VEL
LIN {X 0,Y 355.377,Z 401.98,A -85,B 0,C 180,E1 -22698.921,E2 -22698.921} C_VEL
LIN {X 0,Y 358.077,Z 411.08,A -85,B 0,C 180,E1 -22700.942,E2 -22700.942} C_VEL
LIN {X 0,Y 361.157,Z 423.112,A -85,B 0,C 180,E1 -22703.145,E2 -22703.145} C_VEL
LIN {X 0,Y 340.281,Z 572.859,A -85,B 0,C 180,E1 -22707.147,E2 -22707.147} C_VEL
LIN {X 0,Y 335.702,Z 633.53,A -85,B 0,C 180,E1 -22708.43,E2 -22708.43} C_VEL
LIN {X 0,Y 331.735,Z 667.995,A -85,B 0,C 180,E1 -22709.339,E2 -22709.339} C_VEL
LIN {X 0,Y 326.687,Z 701.265,A -85,B 0,C 180,E1 -22710.44,E2 -22710.44} C_VEL
LIN {X 0,Y 321.248,Z 731.398,A -85,B 0,C 180,E1 -22711.68,E2 -22711.68} C_VEL
LIN {X 0,Y 315.648,Z 758.328,A -85,B 0,C 180,E1 -22713.085,E2 -22713.085} C_VEL
LIN {X 0,Y 309.661,Z 785.042,A -85,B 0,C 180,E1 -22714.737,E2 -22714.737} C_VEL
LIN {X 0,Y 304.091,Z 807.531,A -85,B 0,C 180,E1 -22716.424,E2 -22716.424} C_VEL
LIN {X 0,Y 298.703,Z 825.778,A -85,B 0,C 180,E1 -22718.127,E2 -22718.127} C_VEL
LIN {X 0,Y 292.289,Z 844.528,A -85,B 0,C 180,E1 -22720.283,E2 -22720.283} C_VEL
LIN {X 0,Y 285.621,Z 862.049,A -85,B 0,C 180,E1 -22722.777,E2 -22722.777} C_VEL
LIN {X 0,Y 278.897,Z 878.424,A -85,B 0,C 180,E1 -22725.645,E2 -22725.645} C_VEL
LIN {X 0,Y 272.274,Z 893.536,A -85,B 0,C 180,E1 -22728.902,E2 -22728.902} C_VEL
LIN {X 0,Y 266.16,Z 907.221,A -85,B 0,C 180,E1 -22732.513,E2 -22732.513} C_VEL
LIN {X 0,Y 260.454,Z 920.133,A -85,B 0,C 180,E1 -22736.703,E2 -22736.703} C_VEL
LIN {X 0,Y 256.003,Z 930.92,A -85,B 0,C 180,E1 -22741.033,E2 -22741.033} C_VEL
LIN {X 0,Y 252.644,Z 940.22,A -85,B 0,C 180,E1 -22745.695,E2 -22745.695} C_VEL
LIN {X 0,Y 250.518,Z 947.999,A -85,B 0,C 180,E1 -22750.654,E2 -22750.654} C_VEL
LIN {X 0,Y 249.63,Z 954.104,A -85,B 0,C 180,E1 -22755.774,E2 -22755.774} C_VEL
LIN {X 0,Y 249.741,Z 958.149,A -85,B 0,C 180,E1 -22760.552,E2 -22760.552} C_VEL
LIN {X 0,Y 250.282,Z 960.475,A -85,B 0,C 180,E1 -22764.958,E2 -22764.958} C_VEL
LIN {X 0,Y 250.644,Z 961.382,A -85,B 0,C 180,E1 -22768.857,E2 -22768.857} C_VEL
LIN {X 0,Y 250.335,Z 962.567,A -85,B 0,C 180,E1 -22772.747,E2 -22772.747} C_VEL
LIN {X 0,Y 249.626,Z 962.76,A -85,B 0,C 180,E1 -22777.133,E2 -22777.133} C_VEL
LIN {X 0,Y 249.152,Z 961.367,A -85,B 0,C 180,E1 -22782.281,E2 -22782.281} C_VEL
LIN {X 0,Y 249.664,Z 958.616,A -85,B 0,C 180,E1 -22787.48,E2 -22787.48} C_VEL
LIN {X 0,Y 252.286,Z 953.52,A -85,B 0,C 180,E1 -22793.845,E2 -22793.845} C_VEL
LIN {X 0,Y 257.451,Z 946.724,A -85,B 0,C 180,E1 -22799.992,E2 -22799.992} C_VEL
LIN {X 0,Y 266.746,Z 937.029,A -85,B 0,C 180,E1 -22806.662,E2 -22806.662} C_VEL
LIN {X 0,Y 279.704,Z 925.495,A -85,B 0,C 180,E1 -22812.783,E2 -22812.783} C_VEL
LIN {X 0,Y 295.674,Z 912.532,A -85,B 0,C 180,E1 -22818.072,E2 -22818.072} C_VEL
LIN {X 0,Y 314.698,Z 898.105,A -85,B 0,C 180,E1 -22822.637,E2 -22822.637} C_VEL
LIN {X 0,Y 316.287,Z 896.898,A -85,B 0,C 180,E1 -22823.01,E2 -22823.01} C_VEL
LIN {X 0,Y 300.022,Z 904.665,A -85,B 0,C 180,E1 -22826.774,E2 -22826.774} C_VEL
LIN {X 0,Y 286.291,Z 910.541,A -85,B 0,C 180,E1 -22830.957,E2 -22830.957} C_VEL
LIN {X 0,Y 275.39,Z 914.302,A -85,B 0,C 180,E1 -22835.32,E2 -22835.32} C_VEL
LIN {X 0,Y 266.856,Z 916.048,A -85,B 0,C 180,E1 -22839.835,E2 -22839.835} C_VEL
LIN {X 0,Y 260.728,Z 915.908,A -85,B 0,C 180,E1 -22844.2,E2 -22844.2} C_VEL
LIN {X 0,Y 256.348,Z 914.113,A -85,B 0,C 180,E1 -22848.526,E2 -22848.526} C_VEL
LIN {X 0,Y 253.172,Z 910.306,A -85,B 0,C 180,E1 -22853.195,E2 -22853.195} C_VEL
LIN {X 0,Y 251.366,Z 904.758,A -85,B 0,C 180,E1 -22857.72,E2 -22857.72} C_VEL
LIN {X 0,Y 250.557,Z 897.616,A -85,B 0,C 180,E1 -22862.058,E2 -22862.058} C_VEL
LIN {X 0,Y 250.486,Z 889.011,A -85,B 0,C 180,E1 -22866.187,E2 -22866.187} C_VEL
LIN {X 0,Y 251.021,Z 879.044,A -85,B 0,C 180,E1 -22870.094,E2 -22870.094} C_VEL
LIN {X 0,Y 252.205,Z 867.049,A -85,B 0,C 180,E1 -22873.995,E2 -22873.995} C_VEL
LIN {X 0,Y 254.132,Z 852.773,A -85,B 0,C 180,E1 -22877.872,E2 -22877.872} C_VEL
LIN {X 0,Y 256.667,Z 836.908,A -85,B 0,C 180,E1 -22881.481,E2 -22881.481} C_VEL
LIN {X 0,Y 259.61,Z 820.001,A -85,B 0,C 180,E1 -22884.702,E2 -22884.702} C_VEL
LIN {X 0,Y 263.068,Z 800.909,A -85,B 0,C 180,E1 -22887.75,E2 -22887.75} C_VEL
LIN {X 0,Y 265.919,Z 785.589,A -85,B 0,C 180,E1 -22889.882,E2 -22889.882} C_VEL
LIN {X 0,Y 267.556,Z 785.32,A -85,B 0,C 180,E1 -22890.547,E2 -22890.547} C_VEL
LIN {X 0,Y 270.953,Z 783.098,A -85,B 0,C 180,E1 -22891.355,E2 -22891.355} C_VEL
LIN {X 0,Y 273.496,Z 780.839,A -85,B 0,C 180,E1 -22891.767,E2 -22891.767} C_VEL
LIN {X 0,Y 277.266,Z 778.882,A -85,B 0,C 180,E1 -22892.748,E2 -22892.748} C_VEL
LIN {X 0,Y 282.111,Z 774.981,A -85,B 0,C 180,E1 -22893.567,E2 -22893.567} C_VEL
LIN {X 0,Y 283.627,Z 773.906,A -85,B 0,C 180,E1 -22893.849,E2 -22893.849} C_VEL
LIN {X 0,Y 288,Z 771.06,A -85,B 0,C 180,E1 -22894.707,E2 -22894.707} C_VEL
LIN {X 0,Y 293.595,Z 766.149,A -85,B 0,C 180,E1 -22895.486,E2 -22895.486} C_VEL
LIN {X 0,Y 299.852,Z 761.546,A -85,B 0,C 180,E1 -22896.52,E2 -22896.52} C_VEL
LIN {X 0,Y 305.844,Z 755.879,A -85,B 0,C 180,E1 -22897.216,E2 -22897.216} C_VEL
LIN {X 0,Y 307.636,Z 754.215,A -85,B 0,C 180,E1 -22897.43,E2 -22897.43} C_VEL
LIN {X 0,Y 313.568,Z 749.089,A -85,B 0,C 180,E1 -22898.216,E2 -22898.216} C_VEL
LIN {X 0,Y 319.861,Z 742.293,A -85,B 0,C 180,E1 -22898.812,E2 -22898.812} C_VEL
LIN {X 0,Y 322.837,Z 738.833,A -85,B 0,C 180,E1 -22899.071,E2 -22899.071} C_VEL
LIN {X 0,Y 323.024,Z 738.715,A -85,B 0,C 180,E1 -22899.101,E2 -22899.101} C_VEL
LIN {X 0,Y 317.433,Z 758.321,A -85,B 0,C 180,E1 -22900.695,E2 -22900.695} C_VEL
LIN {X 0,Y 311.041,Z 777.243,A -85,B 0,C 180,E1 -22902.595,E2 -22902.595} C_VEL
LIN {X 0,Y 303.938,Z 795.536,A -85,B 0,C 180,E1 -22904.85,E2 -22904.85} C_VEL
LIN {X 0,Y 296.452,Z 812.676,A -85,B 0,C 180,E1 -22907.448,E2 -22907.448} C_VEL
LIN {X 0,Y 288.766,Z 828.6,A -85,B 0,C 180,E1 -22910.422,E2 -22910.422} C_VEL
LIN {X 0,Y 281.516,Z 842.523,A -85,B 0,C 180,E1 -22913.619,E2 -22913.619} C_VEL
LIN {X 0,Y 274.282,Z 855.624,A -85,B 0,C 180,E1 -22917.348,E2 -22917.348} C_VEL
LIN {X 0,Y 267.984,Z 866.636,A -85,B 0,C 180,E1 -22921.262,E2 -22921.262} C_VEL
LIN {X 0,Y 262.335,Z 876.359,A -85,B 0,C 180,E1 -22925.637,E2 -22925.637} C_VEL
LIN {X 0,Y 257.98,Z 883.994,A -85,B 0,C 180,E1 -22930.057,E2 -22930.057} C_VEL
LIN {X 0,Y 254.652,Z 890.073,A -85,B 0,C 180,E1 -22934.747,E2 -22934.747} C_VEL
LIN {X 0,Y 252.375,Z 894.573,A -85,B 0,C 180,E1 -22939.73,E2 -22939.73} C_VEL
LIN {X 0,Y 251.201,Z 897.161,A -85,B 0,C 180,E1 -22944.518,E2 -22944.518} C_VEL
LIN {X 0,Y 250.779,Z 898.152,A -85,B 0,C 180,E1 -22949.086,E2 -22949.086} C_VEL
LIN {X 0,Y 250.968,Z 897.684,A -85,B 0,C 180,E1 -22953.883,E2 -22953.883} C_VEL
LIN {X 0,Y 251.874,Z 895.635,A -85,B 0,C 180,E1 -22958.702,E2 -22958.702} C_VEL
LIN {X 0,Y 253.644,Z 892.014,A -85,B 0,C 180,E1 -22963.449,E2 -22963.449} C_VEL
LIN {X 0,Y 256.519,Z 886.679,A -85,B 0,C 180,E1 -22968.17,E2 -22968.17} C_VEL
LIN {X 0,Y 260.574,Z 879.522,A -85,B 0,C 180,E1 -22972.803,E2 -22972.803} C_VEL
LIN {X 0,Y 265.604,Z 870.883,A -85,B 0,C 180,E1 -22977.098,E2 -22977.098} C_VEL
LIN {X 0,Y 271.76,Z 860.242,A -85,B 0,C 180,E1 -22981.251,E2 -22981.251} C_VEL
LIN {X 0,Y 278.629,Z 848.026,A -85,B 0,C 180,E1 -22985.042,E2 -22985.042} C_VEL
LIN {X 0,Y 285.817,Z 834.602,A -85,B 0,C 180,E1 -22988.405,E2 -22988.405} C_VEL
LIN {X 0,Y 293.217,Z 819.817,A -85,B 0,C 180,E1 -22991.418,E2 -22991.418} C_VEL
LIN {X 0,Y 300.501,Z 803.968,A -85,B 0,C 180,E1 -22994.061,E2 -22994.061} C_VEL
LIN {X 0,Y 307.713,Z 786.538,A -85,B 0,C 180,E1 -22996.437,E2 -22996.437} C_VEL
LIN {X 0,Y 314.433,Z 768.065,A -85,B 0,C 180,E1 -22998.494,E2 -22998.494} C_VEL
LIN {X 0,Y 320.382,Z 749.009,A -85,B 0,C 180,E1 -23000.223,E2 -23000.223} C_VEL
LIN {X 0,Y 325.424,Z 729.786,A -85,B 0,C 180,E1 -23001.635,E2 -23001.635} C_VEL
LIN {X 0,Y 329.778,Z 708.764,A -85,B 0,C 180,E1 -23002.866,E2 -23002.866} C_VEL
LIN {X 0,Y 336.016,Z 670.139,A -85,B 0,C 180,E1 -23004.557,E2 -23004.557} C_VEL
LIN {X 0,Y 342.419,Z 630.14,A -85,B 0,C 180,E1 -23005.924,E2 -23005.924} C_VEL
LIN {X 0,Y 346.295,Z 605.133,A -85,B 0,C 180,E1 -23006.631,E2 -23006.631} C_VEL
LIN {X 0,Y 346.885,Z 597.673,A -85,B 0,C 180,E1 -23006.975,E2 -23006.975} C_VEL
LIN {X 0,Y 346.368,Z 578.131,A -85,B 0,C 180,E1 -23008.35,E2 -23008.35} C_VEL
LIN {X 0,Y 346.837,Z 571.682,A -85,B 0,C 180,E1 -23008.613,E2 -23008.613} C_VEL
LIN {X 0,Y 352.341,Z 523.727,A -85,B 0,C 180,E1 -23009.647,E2 -23009.647} C_VEL
LIN {X 0,Y 358.549,Z 453.065,A -85,B 0,C 180,E1 -23010.937,E2 -23010.937} C_VEL
LIN {X 0,Y 364.031,Z 430.052,A -85,B 0,C 180,E1 -23011.629,E2 -23011.629} C_VEL
LIN {X 0,Y 360.047,Z 416.391,A -85,B 0,C 180,E1 -23014.68,E2 -23014.68} C_VEL
LIN {X 0,Y 356.323,Z 404.78,A -85,B 0,C 180,E1 -23017.796,E2 -23017.796} C_VEL
LIN {X 0,Y 352.921,Z 395.214,A -85,B 0,C 180,E1 -23020.856,E2 -23020.856} C_VEL
LIN {X 0,Y 349.976,Z 387.363,A -85,B 0,C 180,E1 -23023.911,E2 -23023.911} C_VEL
LIN {X 0,Y 347.406,Z 380.655,A -85,B 0,C 180,E1 -23027.111,E2 -23027.111} C_VEL
LIN {X 0,Y 345.934,Z 376.873,A -85,B 0,C 180,E1 -23029.34,E2 -23029.34} C_VEL
LIN {X 0,Y 344.819,Z 373.303,A -85,B 0,C 180,E1 -23031.831,E2 -23031.831} C_VEL
LIN {X 0,Y 343.577,Z 369.463,A -85,B 0,C 180,E1 -23035.493,E2 -23035.493} C_VEL
LIN {X 0,Y 343.43,Z 368.82,A -85,B 0,C 180,E1 -23036.495,E2 -23036.495} C_VEL
LIN {X 0,Y 343.479,Z 367.699,A -85,B 0,C 180,E1 -23041.668,E2 -23041.668} C_VEL
LIN {X 0,Y 345.279,Z 368.86,A -85,B 0,C 180,E1 -23046.318,E2 -23046.318} C_VEL
LIN {X 0,Y 345.488,Z 369.332,A -85,B 0,C 180,E1 -23046.731,E2 -23046.731} C_VEL
LIN {X 0,Y 346.364,Z 378.658,A -85,B 0,C 180,E1 -23049.974,E2 -23049.974} C_VEL
LIN {X 0,Y 348.175,Z 390.05,A -85,B 0,C 180,E1 -23053.494,E2 -23053.494} C_VEL
LIN {X 0,Y 352.845,Z 408.971,A -85,B 0,C 180,E1 -23058.419,E2 -23058.419} C_VEL
LIN {X 0,Y 355.205,Z 417.496,A -85,B 0,C 180,E1 -23060.322,E2 -23060.322} C_VEL
LIN {X 0,Y 357.47,Z 426.949,A -85,B 0,C 180,E1 -23062.061,E2 -23062.061} C_VEL
LIN {X 0,Y 336.817,Z 569.861,A -85,B 0,C 180,E1 -23065.874,E2 -23065.874} C_VEL
LIN {X 0,Y 332.163,Z 629.931,A -85,B 0,C 180,E1 -23067.145,E2 -23067.145} C_VEL
LIN {X 0,Y 328.077,Z 664.549,A -85,B 0,C 180,E1 -23068.042,E2 -23068.042} C_VEL
LIN {X 0,Y 322.786,Z 698.857,A -85,B 0,C 180,E1 -23069.161,E2 -23069.161} C_VEL
LIN {X 0,Y 316.896,Z 730.284,A -85,B 0,C 180,E1 -23070.439,E2 -23070.439} C_VEL
LIN {X 0,Y 311.115,Z 757.419,A -85,B 0,C 180,E1 -23071.839,E2 -23071.839} C_VEL
LIN {X 0,Y 304.372,Z 786.191,A -85,B 0,C 180,E1 -23073.637,E2 -23073.637} C_VEL
LIN {X 0,Y 299.425,Z 805.619,A -85,B 0,C 180,E1 -23075.1,E2 -23075.1} C_VEL
LIN {X 0,Y 293.873,Z 823.687,A -85,B 0,C 180,E1 -23076.764,E2 -23076.764} C_VEL
LIN {X 0,Y 287.194,Z 842.545,A -85,B 0,C 180,E1 -23078.918,E2 -23078.918} C_VEL
LIN {X 0,Y 280.407,Z 859.77,A -85,B 0,C 180,E1 -23081.357,E2 -23081.357} C_VEL
LIN {X 0,Y 273.402,Z 876.134,A -85,B 0,C 180,E1 -23084.208,E2 -23084.208} C_VEL
LIN {X 0,Y 266.367,Z 891.442,A -85,B 0,C 180,E1 -23087.493,E2 -23087.493} C_VEL
LIN {X 0,Y 259.868,Z 905.271,A -85,B 0,C 180,E1 -23091.158,E2 -23091.158} C_VEL
LIN {X 0,Y 253.731,Z 918.322,A -85,B 0,C 180,E1 -23095.426,E2 -23095.426} C_VEL
LIN {X 0,Y 248.904,Z 929.249,A -85,B 0,C 180,E1 -23099.858,E2 -23099.858} C_VEL
LIN {X 0,Y 245.191,Z 938.697,A -85,B 0,C 180,E1 -23104.647,E2 -23104.647} C_VEL
LIN {X 0,Y 242.779,Z 946.583,A -85,B 0,C 180,E1 -23109.76,E2 -23109.76} C_VEL
LIN {X 0,Y 241.703,Z 952.882,A -85,B 0,C 180,E1 -23115.139,E2 -23115.139} C_VEL
LIN {X 0,Y 241.721,Z 956.944,A -85,B 0,C 180,E1 -23119.995,E2 -23119.995} C_VEL
LIN {X 0,Y 242.274,Z 959.368,A -85,B 0,C 180,E1 -23124.553,E2 -23124.553} C_VEL
LIN {X 0,Y 242.69,Z 960.344,A -85,B 0,C 180,E1 -23128.584,E2 -23128.584} C_VEL
LIN {X 0,Y 242.617,Z 960.808,A -85,B 0,C 180,E1 -23131.653,E2 -23131.653} C_VEL
LIN {X 0,Y 241.989,Z 961.423,A -85,B 0,C 180,E1 -23135.691,E2 -23135.691} C_VEL
LIN {X 0,Y 241.324,Z 960.912,A -85,B 0,C 180,E1 -23140.263,E2 -23140.263} C_VEL
LIN {X 0,Y 241.346,Z 959.091,A -85,B 0,C 180,E1 -23145.376,E2 -23145.376} C_VEL
LIN {X 0,Y 243.205,Z 954.97,A -85,B 0,C 180,E1 -23151.971,E2 -23151.971} C_VEL
LIN {X 0,Y 247.543,Z 949.265,A -85,B 0,C 180,E1 -23158.29,E2 -23158.29} C_VEL
LIN {X 0,Y 256.061,Z 940.692,A -85,B 0,C 180,E1 -23165.305,E2 -23165.305} C_VEL
LIN {X 0,Y 268.48,Z 930.238,A -85,B 0,C 180,E1 -23171.809,E2 -23171.809} C_VEL
LIN {X 0,Y 284.499,Z 918.06,A -85,B 0,C 180,E1 -23177.566,E2 -23177.566} C_VEL
LIN {X 0,Y 303.916,Z 904.379,A -85,B 0,C 180,E1 -23182.508,E2 -23182.508} C_VEL
LIN {X 0,Y 306.388,Z 902.677,A -85,B 0,C 180,E1 -23183.062,E2 -23183.062} C_VEL
LIN {X 0,Y 290.077,Z 909.42,A -85,B 0,C 180,E1 -23187.001,E2 -23187.001} C_VEL
LIN {X 0,Y 276.681,Z 914.167,A -85,B 0,C 180,E1 -23191.272,E2 -23191.272} C_VEL
LIN {X 0,Y 266.306,Z 916.874,A -85,B 0,C 180,E1 -23195.606,E2 -23195.606} C_VEL
LIN {X 0,Y 258.186,Z 917.772,A -85,B 0,C 180,E1 -23200.074,E2 -23200.074} C_VEL
LIN {X 0,Y 251.859,Z 916.837,A -85,B 0,C 180,E1 -23204.81,E2 -23204.81} C_VEL
LIN {X 0,Y 247.469,Z 914.048,A -85,B 0,C 180,E1 -23209.524,E2 -23209.524} C_VEL
LIN {X 0,Y 244.669,Z 909.579,A -85,B 0,C 180,E1 -23214.136,E2 -23214.136} C_VEL
LIN {X 0,Y 243.134,Z 903.597,A -85,B 0,C 180,E1 -23218.586,E2 -23218.586} C_VEL
LIN {X 0,Y 242.48,Z 895.781,A -85,B 0,C 180,E1 -23223.073,E2 -23223.073} C_VEL
LIN {X 0,Y 242.581,Z 886.484,A -85,B 0,C 180,E1 -23227.341,E2 -23227.341} C_VEL
LIN {X 0,Y 243.385,Z 875.099,A -85,B 0,C 180,E1 -23231.613,E2 -23231.613} C_VEL
LIN {X 0,Y 244.879,Z 862.174,A -85,B 0,C 180,E1 -23235.634,E2 -23235.634} C_VEL
LIN {X 0,Y 247.165,Z 846.76,A -85,B 0,C 180,E1 -23239.62,E2 -23239.62} C_VEL
LIN {X 0,Y 250.095,Z 829.651,A -85,B 0,C 180,E1 -23243.316,E2 -23243.316} C_VEL
LIN {X 0,Y 253.558,Z 810.82,A -85,B 0,C 180,E1 -23246.715,E2 -23246.715} C_VEL
LIN {X 0,Y 256.349,Z 796.184,A -85,B 0,C 180,E1 -23248.985,E2 -23248.985} C_VEL
LIN {X 0,Y 258.063,Z 795.879,A -85,B 0,C 180,E1 -23249.733,E2 -23249.733} C_VEL
LIN {X 0,Y 261.396,Z 793.79,A -85,B 0,C 180,E1 -23250.581,E2 -23250.581} C_VEL
LIN {X 0,Y 263.426,Z 792.151,A -85,B 0,C 180,E1 -23250.952,E2 -23250.952} C_VEL
LIN {X 0,Y 266.688,Z 790.708,A -85,B 0,C 180,E1 -23251.915,E2 -23251.915} C_VEL
LIN {X 0,Y 271.264,Z 787.43,A -85,B 0,C 180,E1 -23252.81,E2 -23252.81} C_VEL
LIN {X 0,Y 272.706,Z 786.509,A -85,B 0,C 180,E1 -23253.115,E2 -23253.115} C_VEL
LIN {X 0,Y 276.903,Z 784.082,A -85,B 0,C 180,E1 -23254.035,E2 -23254.035} C_VEL
LIN {X 0,Y 281.977,Z 780.134,A -85,B 0,C 180,E1 -23254.814,E2 -23254.814} C_VEL
LIN {X 0,Y 287.29,Z 776.786,A -85,B 0,C 180,E1 -23255.812,E2 -23255.812} C_VEL
LIN {X 0,Y 294.134,Z 771.195,A -85,B 0,C 180,E1 -23256.749,E2 -23256.749} C_VEL
LIN {X 0,Y 300.69,Z 766.466,A -85,B 0,C 180,E1 -23257.724,E2 -23257.724} C_VEL
LIN {X 0,Y 308.157,Z 759.605,A -85,B 0,C 180,E1 -23258.535,E2 -23258.535} C_VEL
LIN {X 0,Y 313.629,Z 755.169,A -85,B 0,C 180,E1 -23259.22,E2 -23259.22} C_VEL
LIN {X 0,Y 307.091,Z 774.598,A -85,B 0,C 180,E1 -23261.096,E2 -23261.096} C_VEL
LIN {X 0,Y 299.717,Z 793.413,A -85,B 0,C 180,E1 -23263.341,E2 -23263.341} C_VEL
LIN {X 0,Y 292.142,Z 810.488,A -85,B 0,C 180,E1 -23265.853,E2 -23265.853} C_VEL
LIN {X 0,Y 284.54,Z 825.999,A -85,B 0,C 180,E1 -23268.651,E2 -23268.651} C_VEL
LIN {X 0,Y 276.841,Z 840.469,A -85,B 0,C 180,E1 -23271.858,E2 -23271.858} C_VEL
LIN {X 0,Y 269.273,Z 853.798,A -85,B 0,C 180,E1 -23275.523,E2 -23275.523} C_VEL
LIN {X 0,Y 262.342,Z 865.452,A -85,B 0,C 180,E1 -23279.541,E2 -23279.541} C_VEL
LIN {X 0,Y 256.338,Z 875.316,A -85,B 0,C 180,E1 -23283.846,E2 -23283.846} C_VEL
LIN {X 0,Y 251.296,Z 883.626,A -85,B 0,C 180,E1 -23288.527,E2 -23288.527} C_VEL
LIN {X 0,Y 247.54,Z 890.026,A -85,B 0,C 180,E1 -23293.334,E2 -23293.334} C_VEL
LIN {X 0,Y 244.982,Z 894.672,A -85,B 0,C 180,E1 -23298.225,E2 -23298.225} C_VEL
LIN {X 0,Y 243.461,Z 897.762,A -85,B 0,C 180,E1 -23303.396,E2 -23303.396} C_VEL
LIN {X 0,Y 242.869,Z 899.092,A -85,B 0,C 180,E1 -23308.348,E2 -23308.348} C_VEL
LIN {X 0,Y 242.961,Z 898.929,A -85,B 0,C 180,E1 -23313.067,E2 -23313.067} C_VEL
LIN {X 0,Y 243.762,Z 897.219,A -85,B 0,C 180,E1 -23318.017,E2 -23318.017} C_VEL
LIN {X 0,Y 245.567,Z 893.689,A -85,B 0,C 180,E1 -23323.18,E2 -23323.18} C_VEL
LIN {X 0,Y 248.612,Z 888.313,A -85,B 0,C 180,E1 -23328.283,E2 -23328.283} C_VEL
LIN {X 0,Y 252.766,Z 881.335,A -85,B 0,C 180,E1 -23333.055,E2 -23333.055} C_VEL
LIN {X 0,Y 258.227,Z 872.413,A -85,B 0,C 180,E1 -23337.688,E2 -23337.688} C_VEL
LIN {X 0,Y 264.619,Z 861.893,A -85,B 0,C 180,E1 -23341.938,E2 -23341.938} C_VEL
LIN {X 0,Y 271.738,Z 849.807,A -85,B 0,C 180,E1 -23345.807,E2 -23345.807} C_VEL
LIN {X 0,Y 279.361,Z 836.154,A -85,B 0,C 180,E1 -23349.31,E2 -23349.31} C_VEL
LIN {X 0,Y 287.198,Z 821.088,A -85,B 0,C 180,E1 -23352.431,E2 -23352.431} C_VEL
LIN {X 0,Y 294.856,Z 804.991,A -85,B 0,C 180,E1 -23355.142,E2 -23355.142} C_VEL
LIN {X 0,Y 302.293,Z 787.594,A -85,B 0,C 180,E1 -23357.528,E2 -23357.528} C_VEL
LIN {X 0,Y 308.95,Z 769.937,A -85,B 0,C 180,E1 -23359.513,E2 -23359.513} C_VEL
LIN {X 0,Y 314.933,Z 751.546,A -85,B 0,C 180,E1 -23361.21,E2 -23361.21} C_VEL
LIN {X 0,Y 320.446,Z 731.196,A -85,B 0,C 180,E1 -23362.719,E2 -23362.719} C_VEL
LIN {X 0,Y 324.897,Z 710.419,A -85,B 0,C 180,E1 -23363.943,E2 -23363.943} C_VEL
LIN {X 0,Y 331.323,Z 672.15,A -85,B 0,C 180,E1 -23365.637,E2 -23365.637} C_VEL
LIN {X 0,Y 337.946,Z 631.963,A -85,B 0,C 180,E1 -23367.021,E2 -23367.021} C_VEL
LIN {X 0,Y 345.288,Z 583.472,A -85,B 0,C 180,E1 -23368.331,E2 -23368.331} C_VEL
LIN {X 0,Y 346.837,Z 571.682,A -85,B 0,C 180,E1 -23368.613,E2 -23368.613} C_VEL
LIN {X 0,Y 347.335,Z 564.174,A -85,B 0,C 180,E1 -23368.935,E2 -23368.935} C_VEL
LIN {X 0,Y 346.657,Z 544.538,A -85,B 0,C 180,E1 -23370.272,E2 -23370.272} C_VEL
LIN {X 0,Y 346.997,Z 538.052,A -85,B 0,C 180,E1 -23370.51,E2 -23370.51} C_VEL
LIN {X 0,Y 352.357,Z 479.814,A -85,B 0,C 180,E1 -23371.595,E2 -23371.595} C_VEL
LIN {X 0,Y 354.602,Z 455.735,A -85,B 0,C 180,E1 -23372.031,E2 -23372.031} C_VEL
LIN {X 0,Y 359.756,Z 433.802,A -85,B 0,C 180,E1 -23372.703,E2 -23372.703} C_VEL
LIN {X 0,Y 355.977,Z 420.386,A -85,B 0,C 180,E1 -23375.833,E2 -23375.833} C_VEL
LIN {X 0,Y 352.347,Z 408.944,A -85,B 0,C 180,E1 -23379.049,E2 -23379.049} C_VEL
LIN {X 0,Y 349.186,Z 399.554,A -85,B 0,C 180,E1 -23382.244,E2 -23382.244} C_VEL
LIN {X 0,Y 346.458,Z 391.969,A -85,B 0,C 180,E1 -23385.458,E2 -23385.458} C_VEL
LIN {X 0,Y 344.769,Z 387.315,A -85,B 0,C 180,E1 -23387.862,E2 -23387.862} C_VEL
LIN {X 0,Y 343.643,Z 384.271,A -85,B 0,C 180,E1 -23389.692,E2 -23389.692} C_VEL
LIN {X 0,Y 342.522,Z 380.827,A -85,B 0,C 180,E1 -23392.114,E2 -23392.114} C_VEL
LIN {X 0,Y 341.574,Z 376.877,A -85,B 0,C 180,E1 -23395.887,E2 -23395.887} C_VEL
LIN {X 0,Y 341.688,Z 375.496,A -85,B 0,C 180,E1 -23401.677,E2 -23401.677} C_VEL
LIN {X 0,Y 343.463,Z 376.678,A -85,B 0,C 180,E1 -23406.309,E2 -23406.309} C_VEL
LIN {X 0,Y 344.276,Z 386.078,A -85,B 0,C 180,E1 -23409.571,E2 -23409.571} C_VEL
LIN {X 0,Y 345.899,Z 396.844,A -85,B 0,C 180,E1 -23412.903,E2 -23412.903} C_VEL
LIN {X 0,Y 350.144,Z 415.442,A -85,B 0,C 180,E1 -23417.792,E2 -23417.792} C_VEL
LIN {X 0,Y 352.332,Z 423.731,A -85,B 0,C 180,E1 -23419.651,E2 -23419.651} C_VEL
LIN {X 0,Y 353.872,Z 430.799,A -85,B 0,C 180,E1 -23420.957,E2 -23420.957} C_VEL
LIN {X 0,Y 333.513,Z 567.002,A -85,B 0,C 180,E1 -23424.578,E2 -23424.578} C_VEL
LIN {X 0,Y 328.621,Z 627.947,A -85,B 0,C 180,E1 -23425.871,E2 -23425.871} C_VEL
LIN {X 0,Y 324.389,Z 662.655,A -85,B 0,C 180,E1 -23426.761,E2 -23426.761} C_VEL
LIN {X 0,Y 319.068,Z 696.214,A -85,B 0,C 180,E1 -23427.843,E2 -23427.843} C_VEL
LIN {X 0,Y 313.154,Z 727.135,A -85,B 0,C 180,E1 -23429.065,E2 -23429.065} C_VEL
LIN {X 0,Y 306.952,Z 755.501,A -85,B 0,C 180,E1 -23430.503,E2 -23430.503} C_VEL
LIN {X 0,Y 299.604,Z 786.015,A -85,B 0,C 180,E1 -23432.397,E2 -23432.397} C_VEL
LIN {X 0,Y 293.809,Z 807.39,A -85,B 0,C 180,E1 -23434.037,E2 -23434.037} C_VEL
LIN {X 0,Y 287.815,Z 825.742,A -85,B 0,C 180,E1 -23435.787,E2 -23435.787} C_VEL
LIN {X 0,Y 280.907,Z 844.161,A -85,B 0,C 180,E1 -23437.961,E2 -23437.961} C_VEL
LIN {X 0,Y 273.611,Z 861.525,A -85,B 0,C 180,E1 -23440.525,E2 -23440.525} C_VEL
LIN {X 0,Y 266.144,Z 877.913,A -85,B 0,C 180,E1 -23443.524,E2 -23443.524} C_VEL
LIN {X 0,Y 258.919,Z 892.811,A -85,B 0,C 180,E1 -23446.879,E2 -23446.879} C_VEL
LIN {X 0,Y 252.232,Z 906.31,A -85,B 0,C 180,E1 -23450.635,E2 -23450.635} C_VEL
LIN {X 0,Y 246.224,Z 918.438,A -85,B 0,C 180,E1 -23454.785,E2 -23454.785} C_VEL
LIN {X 0,Y 241.198,Z 929.146,A -85,B 0,C 180,E1 -23459.343,E2 -23459.343} C_VEL
LIN {X 0,Y 237.18,Z 938.805,A -85,B 0,C 180,E1 -23464.532,E2 -23464.532} C_VEL
LIN {X 0,Y 234.746,Z 946.482,A -85,B 0,C 180,E1 -23469.817,E2 -23469.817} C_VEL
LIN {X 0,Y 233.715,Z 952.415,A -85,B 0,C 180,E1 -23475.215,E2 -23475.215} C_VEL
LIN {X 0,Y 233.795,Z 956.418,A -85,B 0,C 180,E1 -23480.399,E2 -23480.399} C_VEL
LIN {X 0,Y 234.399,Z 958.644,A -85,B 0,C 180,E1 -23485.106,E2 -23485.106} C_VEL
LIN {X 0,Y 234.776,Z 959.382,A -85,B 0,C 180,E1 -23489.024,E2 -23489.024} C_VEL
LIN {X 0,Y 234.655,Z 959.491,A -85,B 0,C 180,E1 -23492.442,E2 -23492.442} C_VEL
LIN {X 0,Y 233.929,Z 960.029,A -85,B 0,C 180,E1 -23496.627,E2 -23496.627} C_VEL
LIN {X 0,Y 233.324,Z 959.466,A -85,B 0,C 180,E1 -23501.369,E2 -23501.369} C_VEL
LIN {X 0,Y 233.566,Z 957.616,A -85,B 0,C 180,E1 -23506.668,E2 -23506.668} C_VEL
LIN {X 0,Y 236.074,Z 953.379,A -85,B 0,C 180,E1 -23513.727,E2 -23513.727} C_VEL
LIN {X 0,Y 241.373,Z 947.552,A -85,B 0,C 180,E1 -23520.357,E2 -23520.357} C_VEL
LIN {X 0,Y 251.549,Z 938.733,A -85,B 0,C 180,E1 -23527.745,E2 -23527.745} C_VEL
LIN {X 0,Y 265.876,Z 928.157,A -85,B 0,C 180,E1 -23534.387,E2 -23534.387} C_VEL
LIN {X 0,Y 283.382,Z 916.29,A -85,B 0,C 180,E1 -23539.967,E2 -23539.967} C_VEL
LIN {X 0,Y 296.308,Z 907.981,A -85,B 0,C 180,E1 -23543.137,E2 -23543.137} C_VEL
LIN {X 0,Y 280.326,Z 913.596,A -85,B 0,C 180,E1 -23547.169,E2 -23547.169} C_VEL
LIN {X 0,Y 267.516,Z 917.249,A -85,B 0,C 180,E1 -23551.417,E2 -23551.417} C_VEL
LIN {X 0,Y 257.188,Z 919.111,A -85,B 0,C 180,E1 -23555.907,E2 -23555.907} C_VEL
LIN {X 0,Y 248.834,Z 919.122,A -85,B 0,C 180,E1 -23560.761,E2 -23560.761} C_VEL
LIN {X 0,Y 242.975,Z 917.338,A -85,B 0,C 180,E1 -23565.462,E2 -23565.462} C_VEL
LIN {X 0,Y 238.945,Z 913.958,A -85,B 0,C 180,E1 -23570.121,E2 -23570.121} C_VEL
LIN {X 0,Y 236.299,Z 908.835,A -85,B 0,C 180,E1 -23574.902,E2 -23574.902} C_VEL
LIN {X 0,Y 234.928,Z 902.216,A -85,B 0,C 180,E1 -23579.512,E2 -23579.512} C_VEL
LIN {X 0,Y 234.446,Z 894.223,A -85,B 0,C 180,E1 -23583.913,E2 -23583.913} C_VEL
LIN {X 0,Y 234.7,Z 884.316,A -85,B 0,C 180,E1 -23588.329,E2 -23588.329} C_VEL
LIN {X 0,Y 235.701,Z 872.242,A -85,B 0,C 180,E1 -23592.744,E2 -23592.744} C_VEL
LIN {X 0,Y 237.448,Z 858.577,A -85,B 0,C 180,E1 -23596.892,E2 -23596.892} C_VEL
LIN {X 0,Y 239.856,Z 843.366,A -85,B 0,C 180,E1 -23600.753,E2 -23600.753} C_VEL
LIN {X 0,Y 242.896,Z 826.279,A -85,B 0,C 180,E1 -23604.382,E2 -23604.382} C_VEL
LIN {X 0,Y 246.544,Z 807.022,A -85,B 0,C 180,E1 -23607.801,E2 -23607.801} C_VEL
LIN {X 0,Y 246.823,Z 806.063,A -85,B 0,C 180,E1 -23608.029,E2 -23608.029} C_VEL
LIN {X 0,Y 248.589,Z 805.719,A -85,B 0,C 180,E1 -23608.86,E2 -23608.86} C_VEL
LIN {X 0,Y 251.85,Z 803.755,A -85,B 0,C 180,E1 -23609.754,E2 -23609.754} C_VEL
LIN {X 0,Y 253.415,Z 802.585,A -85,B 0,C 180,E1 -23610.073,E2 -23610.073} C_VEL
LIN {X 0,Y 256.887,Z 801.096,A -85,B 0,C 180,E1 -23611.177,E2 -23611.177} C_VEL
LIN {X 0,Y 261.355,Z 798.141,A -85,B 0,C 180,E1 -23612.126,E2 -23612.126} C_VEL
LIN {X 0,Y 265.965,Z 795.781,A -85,B 0,C 180,E1 -23613.291,E2 -23613.291} C_VEL
LIN {X 0,Y 270.732,Z 792.531,A -85,B 0,C 180,E1 -23614.151,E2 -23614.151} C_VEL
LIN {X 0,Y 275.815,Z 789.679,A -85,B 0,C 180,E1 -23615.199,E2 -23615.199} C_VEL
LIN {X 0,Y 281.675,Z 785.442,A -85,B 0,C 180,E1 -23616.105,E2 -23616.105} C_VEL
LIN {X 0,Y 288.032,Z 781.326,A -85,B 0,C 180,E1 -23617.16,E2 -23617.16} C_VEL
LIN {X 0,Y 294.281,Z 776.492,A -85,B 0,C 180,E1 -23617.951,E2 -23617.951} C_VEL
LIN {X 0,Y 301.059,Z 771.653,A -85,B 0,C 180,E1 -23618.882,E2 -23618.882} C_VEL
LIN {X 0,Y 304.437,Z 768.801,A -85,B 0,C 180,E1 -23619.247,E2 -23619.247} C_VEL
LIN {X 0,Y 297.401,Z 787.222,A -85,B 0,C 180,E1 -23621.286,E2 -23621.286} C_VEL
LIN {X 0,Y 289.716,Z 804.818,A -85,B 0,C 180,E1 -23623.679,E2 -23623.679} C_VEL
LIN {X 0,Y 281.607,Z 821.407,A -85,B 0,C 180,E1 -23626.462,E2 -23626.462} C_VEL
LIN {X 0,Y 273.828,Z 835.892,A -85,B 0,C 180,E1 -23629.46,E2 -23629.46} C_VEL
LIN {X 0,Y 266.256,Z 849.006,A -85,B 0,C 180,E1 -23632.799,E2 -23632.799} C_VEL
LIN {X 0,Y 259.078,Z 860.781,A -85,B 0,C 180,E1 -23636.503,E2 -23636.503} C_VEL
LIN {X 0,Y 252.194,Z 871.677,A -85,B 0,C 180,E1 -23640.812,E2 -23640.812} C_VEL
LIN {X 0,Y 246.468,Z 880.603,A -85,B 0,C 180,E1 -23645.333,E2 -23645.333} C_VEL
LIN {X 0,Y 241.823,Z 887.928,A -85,B 0,C 180,E1 -23650.181,E2 -23650.181} C_VEL
LIN {X 0,Y 238.462,Z 893.471,A -85,B 0,C 180,E1 -23655.18,E2 -23655.18} C_VEL
LIN {X 0,Y 236.24,Z 897.45,A -85,B 0,C 180,E1 -23660.499,E2 -23660.499} C_VEL
LIN {X 0,Y 235.164,Z 899.596,A -85,B 0,C 180,E1 -23665.61,E2 -23665.61} C_VEL
LIN {X 0,Y 234.899,Z 900.206,A -85,B 0,C 180,E1 -23670.488,E2 -23670.488} C_VEL
LIN {X 0,Y 235.336,Z 899.324,A -85,B 0,C 180,E1 -23675.608,E2 -23675.608} C_VEL
LIN {X 0,Y 236.607,Z 896.831,A -85,B 0,C 180,E1 -23680.716,E2 -23680.716} C_VEL
LIN {X 0,Y 238.961,Z 892.703,A -85,B 0,C 180,E1 -23685.782,E2 -23685.782} C_VEL
LIN {X 0,Y 242.348,Z 887.166,A -85,B 0,C 180,E1 -23690.53,E2 -23690.53} C_VEL
LIN {X 0,Y 246.933,Z 879.968,A -85,B 0,C 180,E1 -23695.161,E2 -23695.161} C_VEL
LIN {X 0,Y 252.733,Z 870.958,A -85,B 0,C 180,E1 -23699.639,E2 -23699.639} C_VEL
LIN {X 0,Y 259.345,Z 860.52,A -85,B 0,C 180,E1 -23703.723,E2 -23703.723} C_VEL
LIN {X 0,Y 266.99,Z 847.977,A -85,B 0,C 180,E1 -23707.621,E2 -23707.621} C_VEL
LIN {X 0,Y 274.638,Z 834.658,A -85,B 0,C 180,E1 -23710.945,E2 -23710.945} C_VEL
LIN {X 0,Y 282.74,Z 819.433,A -85,B 0,C 180,E1 -23714.02,E2 -23714.02} C_VEL
LIN {X 0,Y 290.627,Z 803.132,A -85,B 0,C 180,E1 -23716.69,E2 -23716.69} C_VEL
LIN {X 0,Y 298.105,Z 785.857,A -85,B 0,C 180,E1 -23718.998,E2 -23718.998} C_VEL
LIN {X 0,Y 305.095,Z 767.411,A -85,B 0,C 180,E1 -23721.005,E2 -23721.005} C_VEL
LIN {X 0,Y 311.158,Z 748.674,A -85,B 0,C 180,E1 -23722.665,E2 -23722.665} C_VEL
LIN {X 0,Y 316.591,Z 728.432,A -85,B 0,C 180,E1 -23724.106,E2 -23724.106} C_VEL
LIN {X 0,Y 320.965,Z 707.582,A -85,B 0,C 180,E1 -23725.282,E2 -23725.282} C_VEL
LIN {X 0,Y 327.653,Z 668.819,A -85,B 0,C 180,E1 -23726.957,E2 -23726.957} C_VEL
LIN {X 0,Y 334.631,Z 627.548,A -85,B 0,C 180,E1 -23728.334,E2 -23728.334} C_VEL
LIN {X 0,Y 341.901,Z 579.415,A -85,B 0,C 180,E1 -23729.593,E2 -23729.593} C_VEL
LIN {X 0,Y 346.997,Z 538.052,A -85,B 0,C 180,E1 -23730.51,E2 -23730.51} C_VEL
LIN {X 0,Y 347.35,Z 530.5,A -85,B 0,C 180,E1 -23730.803,E2 -23730.803} C_VEL
LIN {X 0,Y 346.384,Z 510.784,A -85,B 0,C 180,E1 -23732.106,E2 -23732.106} C_VEL
LIN {X 0,Y 346.622,Z 504.272,A -85,B 0,C 180,E1 -23732.333,E2 -23732.333} C_VEL
LIN {X 0,Y 350.786,Z 458.367,A -85,B 0,C 180,E1 -23733.149,E2 -23733.149} C_VEL
LIN {X 0,Y 355.639,Z 437.88,A -85,B 0,C 180,E1 -23733.751,E2 -23733.751} C_VEL
LIN {X 0,Y 352.368,Z 425.709,A -85,B 0,C 180,E1 -23736.681,E2 -23736.681} C_VEL
LIN {X 0,Y 349.155,Z 415.154,A -85,B 0,C 180,E1 -23739.726,E2 -23739.726} C_VEL
LIN {X 0,Y 346.39,Z 406.434,A -85,B 0,C 180,E1 -23742.746,E2 -23742.746} C_VEL
LIN {X 0,Y 343.844,Z 398.992,A -85,B 0,C 180,E1 -23745.947,E2 -23745.947} C_VEL
LIN {X 0,Y 342.325,Z 394.25,A -85,B 0,C 180,E1 -23748.458,E2 -23748.458} C_VEL
LIN {X 0,Y 341.3,Z 391.444,A -85,B 0,C 180,E1 -23750.217,E2 -23750.217} C_VEL
LIN {X 0,Y 340.4,Z 388.391,A -85,B 0,C 180,E1 -23752.404,E2 -23752.404} C_VEL
LIN {X 0,Y 339.526,Z 384.355,A -85,B 0,C 180,E1 -23756.454,E2 -23756.454} C_VEL
LIN {X 0,Y 339.949,Z 383.311,A -85,B 0,C 180,E1 -23762.023,E2 -23762.023} C_VEL
LIN {X 0,Y 341.472,Z 384.468,A -85,B 0,C 180,E1 -23766.051,E2 -23766.051} C_VEL
LIN {X 0,Y 342.19,Z 394.107,A -85,B 0,C 180,E1 -23769.376,E2 -23769.376} C_VEL
LIN {X 0,Y 343.611,Z 403.92,A -85,B 0,C 180,E1 -23772.393,E2 -23772.393} C_VEL
LIN {X 0,Y 347.54,Z 422.084,A -85,B 0,C 180,E1 -23777.195,E2 -23777.195} C_VEL
LIN {X 0,Y 349.46,Z 429.852,A -85,B 0,C 180,E1 -23778.951,E2 -23778.951} C_VEL
LIN {X 0,Y 350.422,Z 434.607,A -85,B 0,C 180,E1 -23779.829,E2 -23779.829} C_VEL
LIN {X 0,Y 330.399,Z 563.948,A -85,B 0,C 180,E1 -23783.254,E2 -23783.254} C_VEL
LIN {X 0,Y 325.235,Z 626.022,A -85,B 0,C 180,E1 -23784.573,E2 -23784.573} C_VEL
LIN {X 0,Y 320.852,Z 660.895,A -85,B 0,C 180,E1 -23785.455,E2 -23785.455} C_VEL
LIN {X 0,Y 315.405,Z 694.246,A -85,B 0,C 180,E1 -23786.518,E2 -23786.518} C_VEL
LIN {X 0,Y 309.434,Z 724.747,A -85,B 0,C 180,E1 -23787.701,E2 -23787.701} C_VEL
LIN {X 0,Y 302.933,Z 753.57,A -85,B 0,C 180,E1 -23789.136,E2 -23789.136} C_VEL
LIN {X 0,Y 295.72,Z 782.923,A -85,B 0,C 180,E1 -23790.927,E2 -23790.927} C_VEL
LIN {X 0,Y 290.179,Z 803.022,A -85,B 0,C 180,E1 -23792.412,E2 -23792.412} C_VEL
LIN {X 0,Y 283.713,Z 822.483,A -85,B 0,C 180,E1 -23794.208,E2 -23794.208} C_VEL
LIN {X 0,Y 276.538,Z 841.161,A -85,B 0,C 180,E1 -23796.369,E2 -23796.369} C_VEL
LIN {X 0,Y 268.902,Z 858.867,A -85,B 0,C 180,E1 -23798.933,E2 -23798.933} C_VEL
LIN {X 0,Y 261.419,Z 874.651,A -85,B 0,C 180,E1 -23801.768,E2 -23801.768} C_VEL
LIN {X 0,Y 253.722,Z 889.849,A -85,B 0,C 180,E1 -23805.137,E2 -23805.137} C_VEL
LIN {X 0,Y 246.148,Z 904.381,A -85,B 0,C 180,E1 -23809.156,E2 -23809.156} C_VEL
LIN {X 0,Y 239.379,Z 917.279,A -85,B 0,C 180,E1 -23813.62,E2 -23813.62} C_VEL
LIN {X 0,Y 233.997,Z 927.995,A -85,B 0,C 180,E1 -23818.292,E2 -23818.292} C_VEL
LIN {X 0,Y 229.81,Z 937.272,A -85,B 0,C 180,E1 -23823.375,E2 -23823.375} C_VEL
LIN {X 0,Y 226.972,Z 945.352,A -85,B 0,C 180,E1 -23829.057,E2 -23829.057} C_VEL
LIN {X 0,Y 225.786,Z 951.275,A -85,B 0,C 180,E1 -23834.591,E2 -23834.591} C_VEL
LIN {X 0,Y 225.772,Z 955.227,A -85,B 0,C 180,E1 -23839.796,E2 -23839.796} C_VEL
LIN {X 0,Y 226.384,Z 957.536,A -85,B 0,C 180,E1 -23844.678,E2 -23844.678} C_VEL
LIN {X 0,Y 226.821,Z 958.36,A -85,B 0,C 180,E1 -23848.737,E2 -23848.737} C_VEL
LIN {X 0,Y 226.729,Z 958.185,A -85,B 0,C 180,E1 -23852.781,E2 -23852.781} C_VEL
LIN {X 0,Y 225.883,Z 958.597,A -85,B 0,C 180,E1 -23857.631,E2 -23857.631} C_VEL
LIN {X 0,Y 225.37,Z 957.858,A -85,B 0,C 180,E1 -23863.078,E2 -23863.078} C_VEL
LIN {X 0,Y 226.13,Z 955.663,A -85,B 0,C 180,E1 -23869.1,E2 -23869.1} C_VEL
LIN {X 0,Y 229.876,Z 951.018,A -85,B 0,C 180,E1 -23876.617,E2 -23876.617} C_VEL
LIN {X 0,Y 237.165,Z 944.592,A -85,B 0,C 180,E1 -23883.844,E2 -23883.844} C_VEL
LIN {X 0,Y 249.299,Z 935.661,A -85,B 0,C 180,E1 -23891.131,E2 -23891.131} C_VEL
LIN {X 0,Y 266.188,Z 924.791,A -85,B 0,C 180,E1 -23897.748,E2 -23897.748} C_VEL
LIN {X 0,Y 286.276,Z 912.738,A -85,B 0,C 180,E1 -23903.188,E2 -23903.188} C_VEL
LIN {X 0,Y 271.104,Z 917.186,A -85,B 0,C 180,E1 -23907.168,E2 -23907.168} C_VEL
LIN {X 0,Y 257.814,Z 920.039,A -85,B 0,C 180,E1 -23911.76,E2 -23911.76} C_VEL
LIN {X 0,Y 247.222,Z 920.953,A -85,B 0,C 180,E1 -23916.649,E2 -23916.649} C_VEL
LIN {X 0,Y 239.471,Z 919.991,A -85,B 0,C 180,E1 -23921.498,E2 -23921.498} C_VEL
LIN {X 0,Y 233.867,Z 917.343,A -85,B 0,C 180,E1 -23926.399,E2 -23926.399} C_VEL
LIN {X 0,Y 229.964,Z 912.881,A -85,B 0,C 180,E1 -23931.499,E2 -23931.499} C_VEL
LIN {X 0,Y 227.69,Z 906.798,A -85,B 0,C 180,E1 -23936.475,E2 -23936.475} C_VEL
LIN {X 0,Y 226.676,Z 899.674,A -85,B 0,C 180,E1 -23941.011,E2 -23941.011} C_VEL
LIN {X 0,Y 226.455,Z 890.778,A -85,B 0,C 180,E1 -23945.574,E2 -23945.574} C_VEL
LIN {X 0,Y 227.003,Z 879.855,A -85,B 0,C 180,E1 -23950.148,E2 -23950.148} C_VEL
LIN {X 0,Y 228.331,Z 867.078,A -85,B 0,C 180,E1 -23954.582,E2 -23954.582} C_VEL
LIN {X 0,Y 230.407,Z 852.761,A -85,B 0,C 180,E1 -23958.732,E2 -23958.732} C_VEL
LIN {X 0,Y 233.226,Z 836.41,A -85,B 0,C 180,E1 -23962.697,E2 -23962.697} C_VEL
LIN {X 0,Y 236.629,Z 818.334,A -85,B 0,C 180,E1 -23966.339,E2 -23966.339} C_VEL
LIN {X 0,Y 237.276,Z 815.294,A -85,B 0,C 180,E1 -23966.937,E2 -23966.937} C_VEL
LIN {X 0,Y 239.193,Z 814.88,A -85,B 0,C 180,E1 -23967.917,E2 -23967.917} C_VEL
LIN {X 0,Y 242.409,Z 812.984,A -85,B 0,C 180,E1 -23968.856,E2 -23968.856} C_VEL
LIN {X 0,Y 243.699,Z 812.239,A -85,B 0,C 180,E1 -23969.226,E2 -23969.226} C_VEL
LIN {X 0,Y 247.112,Z 810.774,A -85,B 0,C 180,E1 -23970.384,E2 -23970.384} C_VEL
LIN {X 0,Y 250.748,Z 808.509,A -85,B 0,C 180,E1 -23971.225,E2 -23971.225} C_VEL
LIN {X 0,Y 255.175,Z 806.438,A -85,B 0,C 180,E1 -23972.468,E2 -23972.468} C_VEL
LIN {X 0,Y 259.649,Z 803.739,A -85,B 0,C 180,E1 -23973.414,E2 -23973.414} C_VEL
LIN {X 0,Y 264.64,Z 801.14,A -85,B 0,C 180,E1 -23974.546,E2 -23974.546} C_VEL
LIN {X 0,Y 269.4,Z 798.093,A -85,B 0,C 180,E1 -23975.381,E2 -23975.381} C_VEL
LIN {X 0,Y 275.506,Z 794.582,A -85,B 0,C 180,E1 -23976.527,E2 -23976.527} C_VEL
LIN {X 0,Y 281.455,Z 790.564,A -85,B 0,C 180,E1 -23977.409,E2 -23977.409} C_VEL
LIN {X 0,Y 288.642,Z 785.947,A -85,B 0,C 180,E1 -23978.474,E2 -23978.474} C_VEL
LIN {X 0,Y 294.44,Z 781.641,A -85,B 0,C 180,E1 -23979.171,E2 -23979.171} C_VEL
LIN {X 0,Y 295.133,Z 781.191,A -85,B 0,C 180,E1 -23979.269,E2 -23979.269} C_VEL
LIN {X 0,Y 287.625,Z 798.765,A -85,B 0,C 180,E1 -23981.482,E2 -23981.482} C_VEL
LIN {X 0,Y 279.607,Z 815.369,A -85,B 0,C 180,E1 -23984.045,E2 -23984.045} C_VEL
LIN {X 0,Y 271.285,Z 830.931,A -85,B 0,C 180,E1 -23987.01,E2 -23987.01} C_VEL
LIN {X 0,Y 263.105,Z 844.964,A -85,B 0,C 180,E1 -23990.323,E2 -23990.323} C_VEL
LIN {X 0,Y 255.273,Z 857.536,A -85,B 0,C 180,E1 -23994.017,E2 -23994.017} C_VEL
LIN {X 0,Y 247.995,Z 868.647,A -85,B 0,C 180,E1 -23998.117,E2 -23998.117} C_VEL
LIN {X 0,Y 241.508,Z 878.284,A -85,B 0,C 180,E1 -24002.641,E2 -24002.641} C_VEL
LIN {X 0,Y 236.274,Z 886.036,A -85,B 0,C 180,E1 -24007.35,E2 -24007.35} C_VEL
LIN {X 0,Y 232.134,Z 892.334,A -85,B 0,C 180,E1 -24012.451,E2 -24012.451} C_VEL
LIN {X 0,Y 229.303,Z 896.881,A -85,B 0,C 180,E1 -24017.662,E2 -24017.662} C_VEL
LIN {X 0,Y 227.654,Z 899.817,A -85,B 0,C 180,E1 -24023.04,E2 -24023.04} C_VEL
LIN {X 0,Y 226.989,Z 901.115,A -85,B 0,C 180,E1 -24028.485,E2 -24028.485} C_VEL
LIN {X 0,Y 227.125,Z 900.87,A -85,B 0,C 180,E1 -24033.533,E2 -24033.533} C_VEL
LIN {X 0,Y 228.019,Z 899.232,A -85,B 0,C 180,E1 -24038.574,E2 -24038.574} C_VEL
LIN {X 0,Y 230.071,Z 895.719,A -85,B 0,C 180,E1 -24044.086,E2 -24044.086} C_VEL
LIN {X 0,Y 233.499,Z 890.361,A -85,B 0,C 180,E1 -24049.512,E2 -24049.512} C_VEL
LIN {X 0,Y 238.149,Z 883.406,A -85,B 0,C 180,E1 -24054.561,E2 -24054.561} C_VEL
LIN {X 0,Y 244.19,Z 874.496,A -85,B 0,C 180,E1 -24059.43,E2 -24059.43} C_VEL
LIN {X 0,Y 251.207,Z 863.989,A -85,B 0,C 180,E1 -24063.865,E2 -24063.865} C_VEL
LIN {X 0,Y 258.967,Z 851.916,A -85,B 0,C 180,E1 -24067.873,E2 -24067.873} C_VEL
LIN {X 0,Y 266.745,Z 839.131,A -85,B 0,C 180,E1 -24071.279,E2 -24071.279} C_VEL
LIN {X 0,Y 275.248,Z 824.016,A -85,B 0,C 180,E1 -24074.516,E2 -24074.516} C_VEL
LIN {X 0,Y 283.297,Z 808.339,A -85,B 0,C 180,E1 -24077.234,E2 -24077.234} C_VEL
LIN {X 0,Y 291.225,Z 791.102,A -85,B 0,C 180,E1 -24079.66,E2 -24079.66} C_VEL
LIN {X 0,Y 298.585,Z 772.846,A -85,B 0,C 180,E1 -24081.747,E2 -24081.747} C_VEL
LIN {X 0,Y 304.934,Z 754.573,A -85,B 0,C 180,E1 -24083.452,E2 -24083.452} C_VEL
LIN {X 0,Y 310.474,Z 735.613,A -85,B 0,C 180,E1 -24084.886,E2 -24084.886} C_VEL
LIN {X 0,Y 315.348,Z 714.589,A -85,B 0,C 180,E1 -24086.154,E2 -24086.154} C_VEL
LIN {X 0,Y 321.971,Z 677.886,A -85,B 0,C 180,E1 -24087.817,E2 -24087.817} C_VEL
LIN {X 0,Y 328.759,Z 639.028,A -85,B 0,C 180,E1 -24089.195,E2 -24089.195} C_VEL
LIN {X 0,Y 336.258,Z 592.73,A -85,B 0,C 180,E1 -24090.464,E2 -24090.464} C_VEL
LIN {X 0,Y 342.47,Z 545.544,A -85,B 0,C 180,E1 -24091.538,E2 -24091.538} C_VEL
LIN {X 0,Y 346.622,Z 504.272,A -85,B 0,C 180,E1 -24092.333,E2 -24092.333} C_VEL
LIN {X 0,Y 346.829,Z 496.694,A -85,B 0,C 180,E1 -24092.612,E2 -24092.612} C_VEL
LIN {X 0,Y 345.786,Z 476.924,A -85,B 0,C 180,E1 -24093.892,E2 -24093.892} C_VEL
LIN {X 0,Y 346.043,Z 470.407,A -85,B 0,C 180,E1 -24094.114,E2 -24094.114} C_VEL
LIN {X 0,Y 347.16,Z 460.863,A -85,B 0,C 180,E1 -24094.297,E2 -24094.297} C_VEL
LIN {X 0,Y 351.671,Z 441.871,A -85,B 0,C 180,E1 -24094.845,E2 -24094.845} C_VEL
LIN {X 0,Y 348.557,Z 429.987,A -85,B 0,C 180,E1 -24097.838,E2 -24097.838} C_VEL
LIN {X 0,Y 345.457,Z 419.294,A -85,B 0,C 180,E1 -24101.084,E2 -24101.084} C_VEL
LIN {X 0,Y 342.728,Z 410.383,A -85,B 0,C 180,E1 -24104.431,E2 -24104.431} C_VEL
LIN {X 0,Y 340.438,Z 403.169,A -85,B 0,C 180,E1 -24107.878,E2 -24107.878} C_VEL
LIN {X 0,Y 339.23,Z 399.196,A -85,B 0,C 180,E1 -24110.328,E2 -24110.328} C_VEL
LIN {X 0,Y 338.271,Z 395.951,A -85,B 0,C 180,E1 -24112.698,E2 -24112.698} C_VEL
LIN {X 0,Y 337.59,Z 392.091,A -85,B 0,C 180,E1 -24116.604,E2 -24116.604} C_VEL
LIN {X 0,Y 338.009,Z 391.072,A -85,B 0,C 180,E1 -24122.034,E2 -24122.034} C_VEL
LIN {X 0,Y 339.487,Z 392.138,A -85,B 0,C 180,E1 -24125.747,E2 -24125.747} C_VEL
LIN {X 0,Y 340.126,Z 402.438,A -85,B 0,C 180,E1 -24129.262,E2 -24129.262} C_VEL
LIN {X 0,Y 341.317,Z 411.018,A -85,B 0,C 180,E1 -24131.886,E2 -24131.886} C_VEL
LIN {X 0,Y 344.996,Z 428.89,A -85,B 0,C 180,E1 -24136.631,E2 -24136.631} C_VEL
LIN {X 0,Y 346.692,Z 436.289,A -85,B 0,C 180,E1 -24138.301,E2 -24138.301} C_VEL
LIN {X 0,Y 347.021,Z 438.508,A -85,B 0,C 180,E1 -24138.687,E2 -24138.687} C_VEL
LIN {X 0,Y 327.456,Z 561.023,A -85,B 0,C 180,E1 -24141.907,E2 -24141.907} C_VEL
LIN {X 0,Y 322.042,Z 623.917,A -85,B 0,C 180,E1 -24143.243,E2 -24143.243} C_VEL
LIN {X 0,Y 317.459,Z 659.337,A -85,B 0,C 180,E1 -24144.125,E2 -24144.125} C_VEL
LIN {X 0,Y 311.746,Z 693.302,A -85,B 0,C 180,E1 -24145.196,E2 -24145.196} C_VEL
LIN {X 0,Y 304.7,Z 727.554,A -85,B 0,C 180,E1 -24146.539,E2 -24146.539} C_VEL
LIN {X 0,Y 297.83,Z 757.286,A -85,B 0,C 180,E1 -24148.035,E2 -24148.035} C_VEL
LIN {X 0,Y 289.758,Z 788.404,A -85,B 0,C 180,E1 -24149.987,E2 -24149.987} C_VEL
LIN {X 0,Y 283.881,Z 807.826,A -85,B 0,C 180,E1 -24151.529,E2 -24151.529} C_VEL
LIN {X 0,Y 277.441,Z 825.662,A -85,B 0,C 180,E1 -24153.267,E2 -24153.267} C_VEL
LIN {X 0,Y 269.721,Z 844.322,A -85,B 0,C 180,E1 -24155.54,E2 -24155.54} C_VEL
LIN {X 0,Y 261.879,Z 861.341,A -85,B 0,C 180,E1 -24158.137,E2 -24158.137} C_VEL
LIN {X 0,Y 253.797,Z 877.457,A -85,B 0,C 180,E1 -24161.194,E2 -24161.194} C_VEL
LIN {X 0,Y 245.707,Z 892.542,A -85,B 0,C 180,E1 -24164.75,E2 -24164.75} C_VEL
LIN {X 0,Y 238.201,Z 906.098,A -85,B 0,C 180,E1 -24168.774,E2 -24168.774} C_VEL
LIN {X 0,Y 231.304,Z 918.5,A -85,B 0,C 180,E1 -24173.377,E2 -24173.377} C_VEL
LIN {X 0,Y 225.602,Z 929.356,A -85,B 0,C 180,E1 -24178.467,E2 -24178.467} C_VEL
LIN {X 0,Y 221.317,Z 938.634,A -85,B 0,C 180,E1 -24184.009,E2 -24184.009} C_VEL
LIN {X 0,Y 218.761,Z 945.881,A -85,B 0,C 180,E1 -24189.673,E2 -24189.673} C_VEL
LIN {X 0,Y 217.751,Z 951.329,A -85,B 0,C 180,E1 -24195.371,E2 -24195.371} C_VEL
LIN {X 0,Y 217.911,Z 954.912,A -85,B 0,C 180,E1 -24200.759,E2 -24200.759} C_VEL
LIN {X 0,Y 218.581,Z 956.866,A -85,B 0,C 180,E1 -24205.742,E2 -24205.742} C_VEL
LIN {X 0,Y 218.913,Z 957.435,A -85,B 0,C 180,E1 -24209.738,E2 -24209.738} C_VEL
LIN {X 0,Y 218.663,Z 956.951,A -85,B 0,C 180,E1 -24213.933,E2 -24213.933} C_VEL
LIN {X 0,Y 217.776,Z 957.092,A -85,B 0,C 180,E1 -24219.196,E2 -24219.196} C_VEL
LIN {X 0,Y 217.499,Z 956.197,A -85,B 0,C 180,E1 -24224.919,E2 -24224.919} C_VEL
LIN {X 0,Y 218.932,Z 953.783,A -85,B 0,C 180,E1 -24231.431,E2 -24231.431} C_VEL
LIN {X 0,Y 223.988,Z 948.853,A -85,B 0,C 180,E1 -24239.409,E2 -24239.409} C_VEL
LIN {X 0,Y 233.054,Z 942.206,A -85,B 0,C 180,E1 -24246.917,E2 -24246.917} C_VEL
LIN {X 0,Y 247.522,Z 933.039,A -85,B 0,C 180,E1 -24254.335,E2 -24254.335} C_VEL
LIN {X 0,Y 266.25,Z 922.437,A -85,B 0,C 180,E1 -24260.681,E2 -24260.681} C_VEL
LIN {X 0,Y 276.164,Z 917.011,A -85,B 0,C 180,E1 -24263.244,E2 -24263.244} C_VEL
LIN {X 0,Y 260.678,Z 920.591,A -85,B 0,C 180,E1 -24267.52,E2 -24267.52} C_VEL
LIN {X 0,Y 247.59,Z 922.393,A -85,B 0,C 180,E1 -24272.327,E2 -24272.327} C_VEL
LIN {X 0,Y 237.26,Z 922.254,A -85,B 0,C 180,E1 -24277.449,E2 -24277.449} C_VEL
LIN {X 0,Y 229.826,Z 920.318,A -85,B 0,C 180,E1 -24282.531,E2 -24282.531} C_VEL
LIN {X 0,Y 224.59,Z 916.719,A -85,B 0,C 180,E1 -24287.661,E2 -24287.661} C_VEL
LIN {X 0,Y 221.083,Z 911.282,A -85,B 0,C 180,E1 -24292.986,E2 -24292.986} C_VEL
LIN {X 0,Y 219.198,Z 904.22,A -85,B 0,C 180,E1 -24298.17,E2 -24298.17} C_VEL
LIN {X 0,Y 218.489,Z 896.148,A -85,B 0,C 180,E1 -24302.886,E2 -24302.886} C_VEL
LIN {X 0,Y 218.603,Z 886.203,A -85,B 0,C 180,E1 -24307.623,E2 -24307.623} C_VEL
LIN {X 0,Y 219.538,Z 874.118,A -85,B 0,C 180,E1 -24312.361,E2 -24312.361} C_VEL
LIN {X 0,Y 221.278,Z 860.483,A -85,B 0,C 180,E1 -24316.81,E2 -24316.81} C_VEL
LIN {X 0,Y 223.838,Z 844.818,A -85,B 0,C 180,E1 -24321.075,E2 -24321.075} C_VEL
LIN {X 0,Y 227.068,Z 827.49,A -85,B 0,C 180,E1 -24325.008,E2 -24325.008} C_VEL
LIN {X 0,Y 227.792,Z 823.98,A -85,B 0,C 180,E1 -24325.757,E2 -24325.757} C_VEL
LIN {X 0,Y 229.332,Z 823.711,A -85,B 0,C 180,E1 -24326.685,E2 -24326.685} C_VEL
LIN {X 0,Y 232.306,Z 822.132,A -85,B 0,C 180,E1 -24327.701,E2 -24327.701} C_VEL
LIN {X 0,Y 233.62,Z 821.352,A -85,B 0,C 180,E1 -24328.086,E2 -24328.086} C_VEL
LIN {X 0,Y 236.802,Z 820.097,A -85,B 0,C 180,E1 -24329.328,E2 -24329.328} C_VEL
LIN {X 0,Y 240.216,Z 818.14,A -85,B 0,C 180,E1 -24330.243,E2 -24330.243} C_VEL
LIN {X 0,Y 244.439,Z 816.324,A -85,B 0,C 180,E1 -24331.574,E2 -24331.574} C_VEL
LIN {X 0,Y 248.707,Z 813.984,A -85,B 0,C 180,E1 -24332.597,E2 -24332.597} C_VEL
LIN {X 0,Y 254.451,Z 811.105,A -85,B 0,C 180,E1 -24333.988,E2 -24333.988} C_VEL
LIN {X 0,Y 258.017,Z 809.132,A -85,B 0,C 180,E1 -24334.727,E2 -24334.727} C_VEL
LIN {X 0,Y 263.968,Z 805.958,A -85,B 0,C 180,E1 -24335.954,E2 -24335.954} C_VEL
LIN {X 0,Y 268.061,Z 803.474,A -85,B 0,C 180,E1 -24336.642,E2 -24336.642} C_VEL
LIN {X 0,Y 275.267,Z 799.382,A -85,B 0,C 180,E1 -24337.871,E2 -24337.871} C_VEL
LIN {X 0,Y 280.509,Z 796.003,A -85,B 0,C 180,E1 -24338.594,E2 -24338.594} C_VEL
LIN {X 0,Y 285.552,Z 793.118,A -85,B 0,C 180,E1 -24339.37,E2 -24339.37} C_VEL
LIN {X 0,Y 277.304,Z 810.392,A -85,B 0,C 180,E1 -24341.841,E2 -24341.841} C_VEL
LIN {X 0,Y 268.686,Z 826.509,A -85,B 0,C 180,E1 -24344.701,E2 -24344.701} C_VEL
LIN {X 0,Y 259.94,Z 841.364,A -85,B 0,C 180,E1 -24347.986,E2 -24347.986} C_VEL
LIN {X 0,Y 251.484,Z 854.656,A -85,B 0,C 180,E1 -24351.665,E2 -24351.665} C_VEL
LIN {X 0,Y 243.538,Z 866.423,A -85,B 0,C 180,E1 -24355.772,E2 -24355.772} C_VEL
LIN {X 0,Y 236.357,Z 876.652,A -85,B 0,C 180,E1 -24360.333,E2 -24360.333} C_VEL
LIN {X 0,Y 230.446,Z 884.952,A -85,B 0,C 180,E1 -24365.11,E2 -24365.11} C_VEL
LIN {X 0,Y 225.652,Z 891.77,A -85,B 0,C 180,E1 -24370.32,E2 -24370.32} C_VEL
LIN {X 0,Y 222.258,Z 896.813,A -85,B 0,C 180,E1 -24375.674,E2 -24375.674} C_VEL
LIN {X 0,Y 220.105,Z 900.288,A -85,B 0,C 180,E1 -24381.378,E2 -24381.378} C_VEL
LIN {X 0,Y 219.163,Z 901.958,A -85,B 0,C 180,E1 -24386.861,E2 -24386.861} C_VEL
LIN {X 0,Y 219.078,Z 902.088,A -85,B 0,C 180,E1 -24392.092,E2 -24392.092} C_VEL
LIN {X 0,Y 219.828,Z 900.735,A -85,B 0,C 180,E1 -24397.58,E2 -24397.58} C_VEL
LIN {X 0,Y 221.607,Z 897.812,A -85,B 0,C 180,E1 -24403.038,E2 -24403.038} C_VEL
